// TwinCAT 3 PLC project NOTT_CRYO
// ProgramVersion: 3.1.4026.22
// CompilerDefines: VISU_USEPROPERTYINFO
// libraries:
//   ESO Cryo HMI Library, * (ESO)
//   ESO LDC Comm Common Library, * (ESO)
//   ESO LDC Comm Tcp Library, * (ESO)
//   ESO LDC Cryo Library, * (ESO)
//   METIS Cryo PLC, * (KU Leuven)
//   METIS Fuse Library, * (KU Leuven)
//   Tc2_ControllerToolbox, * (Beckhoff Automation GmbH)
//   Tc2_Standard, * (Beckhoff Automation GmbH)
//   Tc2_System, * (Beckhoff Automation GmbH)
//   Tc2_Utilities, * (Beckhoff Automation GmbH)
//   Tc3_EventLogger, * (Beckhoff Automation GmbH)
//   VisuDialogs
// project tree:
//   DUTs/Enumerations/CoolDOwn/ E_NOTT_CRYO_COOLDOWN_STATE.TcDUT
//   DUTs/Enumerations/WarmUP/ E_NOTT_CRYO_WARMUP_STATE.TcDUT
//   DUTs/Enumerations/ E_NOTT_CRYO_CTRL_CMD.TcDUT, E_NOTT_CRYO_CTRL_STATE.TcDUT, E_NOTT_CRYO_HEATER_CTRL.TcDUT
//   DUTs/Enumerations/TCtrl/ T_NOTT_CTRL_LOOP_CTRL.TcDUT
//   DUTs/Enumerations/TempVote/ E_ALL_NOTT_TEMPERATURES.TcDUT
//   DUTs/Structures/CoolDown/ T_NOTT_CRYO_COOLDOWN_CFG.TcDUT, T_NOTT_CRYO_COOLDOWN_CTRL.TcDUT, T_NOTT_CRYO_COOLDOWN_STAT.TcDUT
//   DUTs/Structures/Fan/ T_NOTT_FAN_CFG.TcDUT, T_NOTT_FAN_CTRL.TcDUT, T_NOTT_FAN_STAT.TcDUT
//   DUTs/Structures/Nott_Pump/rp/ T_NOTT_PUMPS_STAT.TcDUT, T_NOTT_PUMP_CFG.TcDUT
//   DUTs/Structures/Nott_Pump/tp/ T_NOTT_PUMP_HIPACE80_CFG.TcDUT, T_NOTT_PUMP_HIPACE80_STAT.TcDUT
//   DUTs/Structures/TempVote/ T_NOTT_TEMP_VOTE_CFG.TcDUT, T_NOTT_CRYO_TEMP_VOTE_STATUS.TcDUT
//   DUTs/Structures/ T_CRYO_EVAC_CFG_50.TcDUT, T_CRYO_EVAC_CTRL_50.TcDUT, T_CRYO_EVAC_STAT_50.TcDUT, T_NOTT_CRYO_CFG.TcDUT, T_NOTT_CRYO_CTRL.TcDUT, T_NOTT_CRYO_DEBUG.TcDUT, T_NOTT_CRYO_EVENTS.TcDUT, T_NOTT_CRYO_STAT.TcDUT, T_NOTT_CRYO_TRIGGERS.TcDUT
//   DUTs/Structures/WarmUp/ T_NOTT_CRYO_WARMUP_CFG.TcDUT, T_NOTT_CRYO_WARMUP_CTRL.TcDUT, T_NOTT_CRYO_WARMUP_STAT.TcDUT
//   / GlobalTextList.TcGTLO, PlcTask.TcTTO, Visualization Manager.TcVMO (not stored)
//   POUs/Devices/Control/ FB_NOTT_CTRL_TEMPERATURE.TcPOU, FB_NOTT_TCTRLs.TcPOU
//   POUs/Devices/Heaters/ FB_NOTT_HEATERS.TcPOU
//   POUs/Devices/Fans/ FB_NOTT_FAN.TcPOU
//   POUs/Devices/ThermalBox/ FB_NOTT_THERMAL_BOX_CONTROL.TcPOU
//   POUs/Devices/NOTT_Pump/Functions/ F_PfeifferExpoNewToLReal.TcPOU (not stored)
//   POUs/Devices/NOTT_Pump/rp/ FB_NOTT_PUMP_HICUBE_80_NEO.TcPOU (not stored)
//   POUs/Devices/NOTT_Pump/tp/ FB_NOTT_PUMP_HIPACE80.TcPOU (not stored)
//   POUs/Devices/Temperatures/ FB_NOTT_TEMPERATURES.TcPOU
//   POUs/Devices/Temp_voters/ FB_NOTT_VOTER.TcPOU, FB_NOTT_VOTERS.TcPOU, FB_NOTT_READ_WRITE_TEMP_VOTE_CONFIG.TcPOU
//   POUs/ FB_NOTT_CRYO_CTRL.TcPOU, MAIN.TcPOU
//   POUs/Routines/CoolDown/ FB_NOTT_CRYO_COOLDOWN.TcPOU
//   POUs/Routines/Evacuation/ FB_NOTT_CRYO_EVAC.TcPOU
//   POUs/Routines/WarmUp/ FB_NOTT_CRYO_WARMUP.TcPOU
//   VISUs/ GUI_TEMPLATE_HIPACE_80.TcVIS, TEMPLATE_NOTT_PUMPS.TcVIS, VISU_BASE_PLATE_HTR.TcVIS, VISU_Detector_Heater.TcVIS, VISU_NOTT_PRESSURES.TcVIS, VISU_NOTT_RP.TcVIS, VISU_NOTT_TP.TcVIS, VISU_PTC_COOLER.TcVIS
// real-time tasks:
//   TASK PlcTask: cycle T#10ms, priority 20, ADS port 350
// I/O:
//   DEVICE Device 1 (EtherCAT), AmsNetId 10.33.179.184.2.1
//     -A1 [EK1200-5000 EtherCAT Power supply (2A E-Bus)]
//       Term 2 (EL6070-0033) [EL6070-0033 1Ch. Licence key terminal, individual licences]
//       A1-N12 (EL4104) [EL4104 4Ch. Ana. Output 0-10V, 16bit]
//       Term 38 (EL2535) [EL2535 2Ch. Pulse Width Current Output (24V, 1A)]
//       Term 39 (EL1084) [EL1084 4Ch. Dig. Input 24V, 3ms, negative]
//       N15_RP_RS485 (EL6021) [EL6021 Interface (RS422/485)]
//       N16_TMP_RS485 (EL6021) [EL6021 Interface (RS422/485)]
//       A1-N5 (EL2068) [EL2068 8Ch. Dig Output 24V, 0.5A]
//       A1-N6_DET_HTR (EL9501) [EL9501 Power supply terminal 0...20 V DC, 0...2 A]
//       A1-N7_DET_SPR_HTR (EL9501) [EL9501 Power supply terminal 0...20 V DC, 0...2 A]
//       A1-N8_SIDECAR_HTR (EL9501) [EL9501 Power supply terminal 0...20 V DC, 0...2 A]
//       A1-N9_P_CHIP_HTR (EL9501) [EL9501 Power supply terminal 0...20 V DC, 0...2 A]
//       A1-N10 (EL2634) [EL2634 4Ch. Relay Output, NO (250V AC / 30V DC)]
//       A1-N11 (EL2634) [EL2634 4Ch. Relay Output, NO (250V AC / 30V DC)]
//       N17_Junction (EK1122) [EK1122 2 port EtherCAT junction]
//     -A2 [EK1101 EtherCAT Coupler (2A E-Bus, ID switch)]
//       A2-N3_T_Sidecar (EL3202-0010) [EL3202-0010 2Ch. Ana. Input PT100 (RTD), High Precision]
//       A2-N4_T_PhotoChip (EL3202-0010) [EL3202-0010 2Ch. Ana. Input PT100 (RTD), High Precision]
//       A2-N5_T_BasePlate (EL3202-0010) [EL3202-0010 2Ch. Ana. Input PT100 (RTD), High Precision]
//       A2-N6_T_Shield (EL3202-0010) [EL3202-0010 2Ch. Ana. Input PT100 (RTD), High Precision]
//       A2-N7_T_FF_Source (EL3202-0010) [EL3202-0010 2Ch. Ana. Input PT100 (RTD), High Precision]
//       A2-N8_T_Environment (EL3218) [EL3218-0000 8Ch. Ana. Input PT100 (RTD)]
//       A2-N9_FF_Current (EL4014) [EL4014 4Ch. Ana. Output 0-20mA, 12bit]
//       A2-N10 (EL3104) [EL3104 4Ch. Ana. Input +/-10V Diff.]
//       A2-N11 (EL3692) [EL3692 2Ch. resistance measurement terminal]
//       A2-N12_Fuse (EL9227-5500) [EL9227-5500 Overcurrent protection 24V DC, 2Ch., max. 10A (sum), adjustable, extended functionalities]
//       A2-N14_LS240 (EL6731) [EL6731 PROFIBUS DP Master]
//       A2-N15_24VPwr (EL9410) [EL9410 E-Bus Power Supplier  (Diagnostics)]
//       A2-N16 (EL1008) [EL1008 8Ch. Dig. Input 24V, 3ms]
//       A2-N17 (EL2612) [EL2612 2Ch. Relay Output, CO (125V AC / 30V DC)]
//       A2-N18_Pump_Start (EL2612) [EL2612 2Ch. Relay Output, CO (125V AC / 30V DC)]
//       A2-N19_PTC_RS485 (EL6021) [EL6021 Interface (RS422/485)]
//       A1-N17_BasePlate_Current_Monitor (EL3681) [EL3681 Digital multimeter terminal]
//       A1-N18_Shield_Current_Monitor (EL3681) [EL3681 Digital multimeter terminal]
//       Term 35 (EL9011) [EL9011 End Terminal]
//   DEVICE Device 6 (NOV-DP-RAM)
//   DEVICE LS240_Det_Temp_Sensors (EL6731), AmsNetId 10.33.179.184.3.1
//     Box 3 (GSD Box) (Model 240 Series) // Vendor: Lake Shore Cryotronics Revision: 1.0
// variable links:
//   NOTT_CRYO/NOTT_CRYO Instance <-> Device 1 (EtherCAT)/-A1/A1-N10 (EL2634)
//     PlcTask Inputs/MAIN.nott_cryo_ctrl.nott_heaters.h_detector.i_nCouplerState <-> InfoData/State
//     PlcTask Outputs/MAIN.nott_cryo_ctrl.nott_heaters.h_detector.io_el95x1.q_bEnable <-> Channel 1/Output
//     PlcTask Outputs/MAIN.nott_cryo_ctrl.nott_heaters.h_detector.io_el95x1.q_bEnable <-> Channel 2/Output
//     PlcTask Outputs/MAIN.nott_cryo_ctrl.nott_heaters.h_detector_spare.io_el95x1.q_bEnable <-> Channel 3/Output
//     PlcTask Outputs/MAIN.nott_cryo_ctrl.nott_heaters.h_detector_spare.io_el95x1.q_bEnable <-> Channel 4/Output
//   NOTT_CRYO/NOTT_CRYO Instance <-> Device 1 (EtherCAT)/-A1/A1-N11 (EL2634)
//     PlcTask Outputs/MAIN.nott_cryo_ctrl.nott_heaters.h_photonic_chip.io_el95x1.q_bEnable <-> Channel 3/Output
//     PlcTask Outputs/MAIN.nott_cryo_ctrl.nott_heaters.h_photonic_chip.io_el95x1.q_bEnable <-> Channel 4/Output
//     PlcTask Outputs/MAIN.nott_cryo_ctrl.nott_heaters.h_sidecar.io_el95x1.q_bEnable <-> Channel 1/Output
//     PlcTask Outputs/MAIN.nott_cryo_ctrl.nott_heaters.h_sidecar.io_el95x1.q_bEnable <-> Channel 2/Output
//   NOTT_CRYO/NOTT_CRYO Instance <-> Device 1 (EtherCAT)/-A1/A1-N12 (EL4104)
//     PlcTask Outputs/MAIN.nott_cryo_ctrl.nott_heaters.h_base_plate.io_cpau60.q_nSetVoltage <-> AO Output Channel 1/SetVoltage_BasePlate_HTR
//     PlcTask Outputs/MAIN.nott_cryo_ctrl.nott_heaters.h_shield.io_cpau60.q_nSetVoltage <-> AO Output Channel 2/SetVoltage_Shield_HTR
//   NOTT_CRYO/NOTT_CRYO Instance <-> Device 1 (EtherCAT)/-A1/A1-N5 (EL2068)
//     PlcTask Inputs/MAIN.nott_cryo_ctrl.evac.PVV1.Actuator.i_nCouplerState <-> InfoData/State
//     PlcTask Inputs/MAIN.nott_cryo_ctrl.nott_heaters.h_base_plate.i_nCouplerState <-> InfoData/State
//     PlcTask Inputs/MAIN.nott_cryo_ctrl.nott_heaters.h_shield.i_nCouplerState <-> InfoData/State
//     PlcTask Outputs/MAIN.nott_cryo_ctrl.evac.PVV1.Actuator.q_bCtrl <-> DOS Outputs Channel 4/PVV1_bCtrl
//     PlcTask Outputs/MAIN.nott_cryo_ctrl.evac.q_bPower_VAGC <-> DOS Outputs Channel 7/Output
//     PlcTask Outputs/MAIN.nott_cryo_ctrl.nott_heaters.h_base_plate.io_cpau60.q_bEnable <-> DOS Outputs Channel 1/bEnable_BasePlate_HTR
//     PlcTask Outputs/MAIN.nott_cryo_ctrl.nott_heaters.h_shield.io_cpau60.q_bEnable <-> DOS Outputs Channel 2/bEnable_Shield_HTR
//   NOTT_CRYO/NOTT_CRYO Instance <-> Device 1 (EtherCAT)/-A1/A1-N6_DET_HTR (EL9501)
//     PlcTask Inputs/MAIN.nott_cryo_ctrl.nott_heaters.h_detector.io_el95x1.i_bError <-> AO Output Status/Status/Error
//     PlcTask Inputs/MAIN.nott_cryo_ctrl.nott_heaters.h_detector.io_el95x1.i_bOutputOverload <-> AO Output Status/Status/Output Overload
//     PlcTask Inputs/MAIN.nott_cryo_ctrl.nott_heaters.h_detector.io_el95x1.i_bOverrange <-> AO Output Status/Status/Overrange
//     PlcTask Inputs/MAIN.nott_cryo_ctrl.nott_heaters.h_detector.io_el95x1.i_bUnderrange <-> AO Output Status/Status/Underrange
//     PlcTask Inputs/MAIN.nott_cryo_ctrl.nott_heaters.h_detector.io_el95x1.i_bWarning <-> AO Output Status/Status/Warning
//     PlcTask Inputs/MAIN.nott_cryo_ctrl.nott_heaters.h_detector.io_el95x1.i_rCurrent <-> AI Output Current Standard (Real32)/io_el95x1.i_rCurrent
//     PlcTask Inputs/MAIN.nott_cryo_ctrl.nott_heaters.h_detector.io_el95x1.i_rVoltage <-> AI Output Voltage Standard (Real32)/Value (Real32)
//     PlcTask Outputs/MAIN.nott_cryo_ctrl.nott_heaters.h_detector.io_el95x1.q_nOutputInterface <-> AO Output Standard (Real32)/Control/Output Interface
//     PlcTask Outputs/MAIN.nott_cryo_ctrl.nott_heaters.h_detector.io_el95x1.q_nOutputOperation <-> AO Output Standard (Real32)/Control/Output Operation
//     PlcTask Outputs/MAIN.nott_cryo_ctrl.nott_heaters.h_detector.io_el95x1.q_rSetVoltage <-> AO Output Standard (Real32)/Value (Real32)
//   NOTT_CRYO/NOTT_CRYO Instance <-> Device 1 (EtherCAT)/-A1/A1-N7_DET_SPR_HTR (EL9501)
//     PlcTask Inputs/MAIN.nott_cryo_ctrl.nott_heaters.h_detector_spare.i_nCouplerState <-> InfoData/State
//     PlcTask Inputs/MAIN.nott_cryo_ctrl.nott_heaters.h_detector_spare.io_el95x1.i_bError <-> AO Output Status/Status/Error
//     PlcTask Inputs/MAIN.nott_cryo_ctrl.nott_heaters.h_detector_spare.io_el95x1.i_bOutputOverload <-> AO Output Status/Status/Output Overload
//     PlcTask Inputs/MAIN.nott_cryo_ctrl.nott_heaters.h_detector_spare.io_el95x1.i_bOverrange <-> AO Output Status/Status/Overrange
//     PlcTask Inputs/MAIN.nott_cryo_ctrl.nott_heaters.h_detector_spare.io_el95x1.i_bUnderrange <-> AO Output Status/Status/Underrange
//     PlcTask Inputs/MAIN.nott_cryo_ctrl.nott_heaters.h_detector_spare.io_el95x1.i_bWarning <-> AO Output Status/Status/Warning
//     PlcTask Inputs/MAIN.nott_cryo_ctrl.nott_heaters.h_detector_spare.io_el95x1.i_rCurrent <-> AI Output Current Standard (Real32)/Value (Real32)
//     PlcTask Inputs/MAIN.nott_cryo_ctrl.nott_heaters.h_detector_spare.io_el95x1.i_rVoltage <-> AI Output Voltage Standard (Real32)/Value (Real32)
//     PlcTask Outputs/MAIN.nott_cryo_ctrl.nott_heaters.h_detector_spare.io_el95x1.q_nOutputInterface <-> AO Output Standard (Real32)/Control/Output Interface
//     PlcTask Outputs/MAIN.nott_cryo_ctrl.nott_heaters.h_detector_spare.io_el95x1.q_nOutputOperation <-> AO Output Standard (Real32)/Control/Output Operation
//     PlcTask Outputs/MAIN.nott_cryo_ctrl.nott_heaters.h_detector_spare.io_el95x1.q_rSetVoltage <-> AO Output Standard (Real32)/Value (Real32)
//   NOTT_CRYO/NOTT_CRYO Instance <-> Device 1 (EtherCAT)/-A1/A1-N8_SIDECAR_HTR (EL9501)
//     PlcTask Inputs/MAIN.nott_cryo_ctrl.nott_heaters.h_sidecar.i_nCouplerState <-> InfoData/State
//     PlcTask Inputs/MAIN.nott_cryo_ctrl.nott_heaters.h_sidecar.io_el95x1.i_bError <-> AO Output Status/Status/Error
//     PlcTask Inputs/MAIN.nott_cryo_ctrl.nott_heaters.h_sidecar.io_el95x1.i_bOutputOverload <-> AO Output Status/Status/Output Overload
//     PlcTask Inputs/MAIN.nott_cryo_ctrl.nott_heaters.h_sidecar.io_el95x1.i_bOverrange <-> AO Output Status/Status/Overrange
//     PlcTask Inputs/MAIN.nott_cryo_ctrl.nott_heaters.h_sidecar.io_el95x1.i_bUnderrange <-> AO Output Status/Status/Underrange
//     PlcTask Inputs/MAIN.nott_cryo_ctrl.nott_heaters.h_sidecar.io_el95x1.i_bWarning <-> AO Output Status/Status/Warning
//     PlcTask Inputs/MAIN.nott_cryo_ctrl.nott_heaters.h_sidecar.io_el95x1.i_rCurrent <-> AI Output Current Standard (Real32)/Value (Real32)
//     PlcTask Inputs/MAIN.nott_cryo_ctrl.nott_heaters.h_sidecar.io_el95x1.i_rVoltage <-> AI Output Voltage Standard (Real32)/Value (Real32)
//     PlcTask Outputs/MAIN.nott_cryo_ctrl.nott_heaters.h_sidecar.io_el95x1.q_nOutputInterface <-> AO Output Standard (Real32)/Control/Output Interface
//     PlcTask Outputs/MAIN.nott_cryo_ctrl.nott_heaters.h_sidecar.io_el95x1.q_nOutputOperation <-> AO Output Standard (Real32)/Control/Output Operation
//     PlcTask Outputs/MAIN.nott_cryo_ctrl.nott_heaters.h_sidecar.io_el95x1.q_rSetVoltage <-> AO Output Standard (Real32)/Value (Real32)
//   NOTT_CRYO/NOTT_CRYO Instance <-> Device 1 (EtherCAT)/-A1/A1-N9_P_CHIP_HTR (EL9501)
//     PlcTask Inputs/MAIN.nott_cryo_ctrl.nott_heaters.h_photonic_chip.i_nCouplerState <-> InfoData/State
//     PlcTask Inputs/MAIN.nott_cryo_ctrl.nott_heaters.h_photonic_chip.io_el95x1.i_bError <-> AO Output Status/Status/Error
//     PlcTask Inputs/MAIN.nott_cryo_ctrl.nott_heaters.h_photonic_chip.io_el95x1.i_bOutputOverload <-> AO Output Status/Status/Output Overload
//     PlcTask Inputs/MAIN.nott_cryo_ctrl.nott_heaters.h_photonic_chip.io_el95x1.i_bOverrange <-> AO Output Status/Status/Overrange
//     PlcTask Inputs/MAIN.nott_cryo_ctrl.nott_heaters.h_photonic_chip.io_el95x1.i_bUnderrange <-> AO Output Status/Status/Underrange
//     PlcTask Inputs/MAIN.nott_cryo_ctrl.nott_heaters.h_photonic_chip.io_el95x1.i_bWarning <-> AO Output Status/Status/Warning
//     PlcTask Inputs/MAIN.nott_cryo_ctrl.nott_heaters.h_photonic_chip.io_el95x1.i_rCurrent <-> AI Output Current Standard (Real32)/Value (Real32)
//     PlcTask Inputs/MAIN.nott_cryo_ctrl.nott_heaters.h_photonic_chip.io_el95x1.i_rVoltage <-> AI Output Voltage Standard (Real32)/Value (Real32)
//     PlcTask Outputs/MAIN.nott_cryo_ctrl.nott_heaters.h_photonic_chip.io_el95x1.q_nOutputInterface <-> AO Output Standard (Real32)/Control/Output Interface
//     PlcTask Outputs/MAIN.nott_cryo_ctrl.nott_heaters.h_photonic_chip.io_el95x1.q_nOutputOperation <-> AO Output Standard (Real32)/Control/Output Operation
//     PlcTask Outputs/MAIN.nott_cryo_ctrl.nott_heaters.h_photonic_chip.io_el95x1.q_rSetVoltage <-> AO Output Standard (Real32)/Value (Real32)
//   NOTT_CRYO/NOTT_CRYO Instance <-> Device 1 (EtherCAT)/-A1/N15_RP_RS485 (EL6021)
//     PlcTask Inputs/MAIN.nott_cryo_ctrl.evac.pump_pvp.comm.COMin_EL60xx/D[{0..21}] <-> COM TxPDO-Map Inputs/Data In {0..21}  (22 links)
//     PlcTask Inputs/MAIN.nott_cryo_ctrl.evac.pump_pvp.comm.COMin_EL60xx/Status <-> COM TxPDO-Map Inputs/Status
//     PlcTask Inputs/MAIN.nott_cryo_ctrl.evac.pump_pvp.comm.i_nCouplerState <-> InfoData/State
//     PlcTask Outputs/MAIN.nott_cryo_ctrl.evac.pump_pvp.comm.COMout_EL60xx/Ctrl <-> COM RxPDO-Map Outputs/Ctrl
//     PlcTask Outputs/MAIN.nott_cryo_ctrl.evac.pump_pvp.comm.COMout_EL60xx/D[{0..21}] <-> COM RxPDO-Map Outputs/Data Out {0..21}  (22 links)
//   NOTT_CRYO/NOTT_CRYO Instance <-> Device 1 (EtherCAT)/-A1/N16_TMP_RS485 (EL6021)
//     PlcTask Inputs/MAIN.nott_cryo_ctrl.evac.pump_tmp.comm.COMin_EL60xx/D[{0..21}] <-> COM TxPDO-Map Inputs/Data In {0..21}  (22 links)
//     PlcTask Inputs/MAIN.nott_cryo_ctrl.evac.pump_tmp.comm.COMin_EL60xx/Status <-> COM TxPDO-Map Inputs/Status
//     PlcTask Inputs/MAIN.nott_cryo_ctrl.evac.pump_tmp.comm.i_nCouplerState <-> InfoData/State
//     PlcTask Outputs/MAIN.nott_cryo_ctrl.evac.pump_tmp.comm.COMout_EL60xx/Ctrl <-> COM RxPDO-Map Outputs/Ctrl
//     PlcTask Outputs/MAIN.nott_cryo_ctrl.evac.pump_tmp.comm.COMout_EL60xx/D[{0..21}] <-> COM RxPDO-Map Outputs/Data Out {0..21}  (22 links)
//   NOTT_CRYO/NOTT_CRYO Instance <-> Device 1 (EtherCAT)/-A1/Term 39 (EL1084)
//     PlcTask Inputs/MAIN.nott_cryo_ctrl.bHMISwitch <-> Channel 2/Input
//   NOTT_CRYO/NOTT_CRYO Instance <-> Device 1 (EtherCAT)/-A2/A1-N17_BasePlate_Current_Monitor (EL3681)
//     PlcTask Inputs/MAIN.nott_cryo_ctrl.nott_heaters.h_base_plate.io_cpau60.i_nActCurrent <-> SAI Inputs/Value
//     PlcTask Inputs/MAIN.nott_cryo_ctrl.nott_heaters.h_base_plate.io_cpau60.i_nStatus <-> SAI Inputs/Status
//   NOTT_CRYO/NOTT_CRYO Instance <-> Device 1 (EtherCAT)/-A2/A1-N18_Shield_Current_Monitor (EL3681)
//     PlcTask Inputs/MAIN.nott_cryo_ctrl.nott_heaters.h_shield.io_cpau60.i_nActCurrent <-> SAI Inputs/Value
//     PlcTask Inputs/MAIN.nott_cryo_ctrl.nott_heaters.h_shield.io_cpau60.i_nStatus <-> SAI Inputs/Status
//   NOTT_CRYO/NOTT_CRYO Instance <-> Device 1 (EtherCAT)/-A2/A2-N10 (EL3104)
//     PlcTask Inputs/MAIN.nott_cryo_ctrl.nott_heaters.h_flat_field.io_flat_field.i_nActVoltage <-> AI Standard Channel 3/Value
//     PlcTask Inputs/MAIN.nott_cryo_ctrl.nott_heaters.h_flat_field.io_flat_field.i_nVoltageStatus <-> AI Standard Channel 3/Status
//     PlcTask Inputs/MAIN.nott_cryo_ctrl.sensor_HPG.i_nStatus <-> AI Standard Channel 2/Status
//     PlcTask Inputs/MAIN.nott_cryo_ctrl.sensor_HPG.i_nValue <-> AI Standard Channel 2/Value
//     PlcTask Inputs/MAIN.nott_cryo_ctrl.sensor_VAGC.i_nStatus <-> AI Standard Channel 1/Status
//     PlcTask Inputs/MAIN.nott_cryo_ctrl.sensor_VAGC.i_nValue <-> AI Standard Channel 1/Value
//   NOTT_CRYO/NOTT_CRYO Instance <-> Device 1 (EtherCAT)/-A2/A2-N16 (EL1008)
//     PlcTask Inputs/MAIN.nott_cryo_ctrl.evac.pump_pvp.i_bError <-> Channel 5/Input
//     PlcTask Inputs/MAIN.nott_cryo_ctrl.evac.pump_tmp.i_bError <-> Channel 8/Input
//     PlcTask Inputs/MAIN.nott_cryo_ctrl.evac.pump_tmp.i_bReady <-> Channel 7/Input
//   NOTT_CRYO/NOTT_CRYO Instance <-> Device 1 (EtherCAT)/-A2/A2-N17 (EL2612)
//     PlcTask Inputs/MAIN.nott_cryo_ctrl.cool_down.cooler.comm.i_nCouplerState <-> InfoData/State
//     PlcTask Outputs/MAIN.nott_cryo_ctrl.bHMIOutEnable <-> Channel 2/Output
//     PlcTask Outputs/MAIN.nott_cryo_ctrl.cool_down.cooler.q_bCtrlStart <-> Channel 1/Output
//   NOTT_CRYO/NOTT_CRYO Instance <-> Device 1 (EtherCAT)/-A2/A2-N18_Pump_Start (EL2612)
//     PlcTask Outputs/MAIN.nott_cryo_ctrl.evac.pump_pvp.q_bStart <-> Channel 1/RP_bEnable
//     PlcTask Outputs/MAIN.nott_cryo_ctrl.evac.pump_tmp.q_bStart <-> Channel 2/TP_bEnable
//   NOTT_CRYO/NOTT_CRYO Instance <-> Device 1 (EtherCAT)/-A2/A2-N19_PTC_RS485 (EL6021)
//     PlcTask Inputs/MAIN.nott_cryo_ctrl.cool_down.cooler.comm.COMin_EL60xx/D[{0..21}] <-> COM TxPDO-Map Inputs/Data In {0..21}  (22 links)
//     PlcTask Inputs/MAIN.nott_cryo_ctrl.cool_down.cooler.comm.COMin_EL60xx/Status <-> COM TxPDO-Map Inputs/Status
//     PlcTask Outputs/MAIN.nott_cryo_ctrl.cool_down.cooler.comm.COMout_EL60xx/Ctrl <-> COM RxPDO-Map Outputs/Ctrl
//     PlcTask Outputs/MAIN.nott_cryo_ctrl.cool_down.cooler.comm.COMout_EL60xx/D[{0..21}] <-> COM RxPDO-Map Outputs/Data Out {0..21}  (22 links)
//   NOTT_CRYO/NOTT_CRYO Instance <-> Device 1 (EtherCAT)/-A2/A2-N3_T_Sidecar (EL3202-0010)
//     PlcTask Inputs/MAIN.nott_cryo_ctrl.nott_temp.t_sidecar_1.i_nStatus <-> RTD Inputs Channel 1/Status
//     PlcTask Inputs/MAIN.nott_cryo_ctrl.nott_temp.t_sidecar_2.i_nStatus <-> RTD Inputs Channel 2/Status
//     PlcTask Inputs/MAIN.nott_cryo_ctrl.nott_temp.t_sidecar_1.i_nValue <-> RTD Inputs Channel 1/Value
//     PlcTask Inputs/MAIN.nott_cryo_ctrl.nott_temp.t_sidecar_2.i_nValue <-> RTD Inputs Channel 2/Value
//   NOTT_CRYO/NOTT_CRYO Instance <-> Device 1 (EtherCAT)/-A2/A2-N4_T_PhotoChip (EL3202-0010)
//     PlcTask Inputs/MAIN.nott_cryo_ctrl.nott_temp.t_photonic_chip_1.i_nStatus <-> RTD Inputs Channel 1/Status
//     PlcTask Inputs/MAIN.nott_cryo_ctrl.nott_temp.t_photonic_chip_2.i_nStatus <-> RTD Inputs Channel 2/Status
//     PlcTask Inputs/MAIN.nott_cryo_ctrl.nott_temp.t_photonic_chip_1.i_nValue <-> RTD Inputs Channel 1/Value
//     PlcTask Inputs/MAIN.nott_cryo_ctrl.nott_temp.t_photonic_chip_2.i_nValue <-> RTD Inputs Channel 2/Value
//   NOTT_CRYO/NOTT_CRYO Instance <-> Device 1 (EtherCAT)/-A2/A2-N5_T_BasePlate (EL3202-0010)
//     PlcTask Inputs/MAIN.nott_cryo_ctrl.nott_temp.t_base_plate_1.i_nStatus <-> RTD Inputs Channel 1/Status
//     PlcTask Inputs/MAIN.nott_cryo_ctrl.nott_temp.t_base_plate_2.i_nStatus <-> RTD Inputs Channel 2/Status
//     PlcTask Inputs/MAIN.nott_cryo_ctrl.nott_temp.t_base_plate_1.i_nValue <-> RTD Inputs Channel 1/Value
//     PlcTask Inputs/MAIN.nott_cryo_ctrl.nott_temp.t_base_plate_2.i_nValue <-> RTD Inputs Channel 2/Value
//   NOTT_CRYO/NOTT_CRYO Instance <-> Device 1 (EtherCAT)/-A2/A2-N6_T_Shield (EL3202-0010)
//     PlcTask Inputs/MAIN.nott_cryo_ctrl.nott_temp.t_shield_1.i_nStatus <-> RTD Inputs Channel 1/Status
//     PlcTask Inputs/MAIN.nott_cryo_ctrl.nott_temp.t_shield_2.i_nStatus <-> RTD Inputs Channel 2/Status
//     PlcTask Inputs/MAIN.nott_cryo_ctrl.nott_temp.t_shield_1.i_nValue <-> RTD Inputs Channel 1/Value
//     PlcTask Inputs/MAIN.nott_cryo_ctrl.nott_temp.t_shield_2.i_nValue <-> RTD Inputs Channel 2/Value
//   NOTT_CRYO/NOTT_CRYO Instance <-> Device 1 (EtherCAT)/-A2/A2-N7_T_FF_Source (EL3202-0010)
//     PlcTask Inputs/MAIN.nott_cryo_ctrl.nott_temp.t_flat_field_1.i_nStatus <-> RTD Inputs Channel 1/Status
//     PlcTask Inputs/MAIN.nott_cryo_ctrl.nott_temp.t_flat_field_2.i_nStatus <-> RTD Inputs Channel 2/Status
//     PlcTask Inputs/MAIN.nott_cryo_ctrl.nott_temp.t_flat_field_1.i_nValue <-> RTD Inputs Channel 1/Value
//     PlcTask Inputs/MAIN.nott_cryo_ctrl.nott_temp.t_flat_field_2.i_nValue <-> RTD Inputs Channel 2/Value
//   NOTT_CRYO/NOTT_CRYO Instance <-> Device 1 (EtherCAT)/-A2/A2-N8_T_Environment (EL3218)
//     PlcTask Inputs/MAIN.nott_cryo_ctrl.nott_temp.t_cabinet_1.i_nStatus <-> RTD Inputs Channel 5/Status
//     PlcTask Inputs/MAIN.nott_cryo_ctrl.nott_temp.t_cabinet_2.i_nStatus <-> RTD Inputs Channel 6/Status
//     PlcTask Inputs/MAIN.nott_cryo_ctrl.nott_temp.t_cabinet_1.i_nValue <-> RTD Inputs Channel 5/Value
//     PlcTask Inputs/MAIN.nott_cryo_ctrl.nott_temp.t_cabinet_2.i_nValue <-> RTD Inputs Channel 6/Value
//     PlcTask Inputs/MAIN.nott_cryo_ctrl.nott_temp.t_thermal_box_{1..4}.i_nStatus <-> RTD Inputs Channel {1..4}/Status  (4 links)
//     PlcTask Inputs/MAIN.nott_cryo_ctrl.nott_temp.t_thermal_box_{1..4}.i_nValue <-> RTD Inputs Channel {1..4}/Value  (4 links)
//   NOTT_CRYO/NOTT_CRYO Instance <-> Device 1 (EtherCAT)/-A2/A2-N9_FF_Current (EL4014)
//     PlcTask Inputs/MAIN.nott_cryo_ctrl.nott_heaters.h_flat_field.i_nCouplerState <-> InfoData/State
//     PlcTask Outputs/MAIN.nott_cryo_ctrl.nott_heaters.h_flat_field.io_flat_field.q_nSetCurrentCh{1..4} <-> AO Outputs Channel {1..4}/Analog output  (4 links)
//   NOTT_CRYO/NOTT_CRYO Instance <-> LS240_Det_Temp_Sensors (EL6731)/Box 3 (GSD Box) (Model 240 Series)
//     PlcTask Inputs/MAIN.nott_cryo_ctrl.nott_temp.t_detector.i_fValue <-> T_DET (Sensor Reading)/Inputs/Sensor Reading_0_0
//     PlcTask Inputs/MAIN.nott_cryo_ctrl.nott_temp.t_detector_spare.i_fValue <-> T_DET_SPARE (Sensor Reading)/Inputs/Sensor Reading_0_0
//   NOTT_CRYO/NOTT_CRYO Instance <-> NOTT_CRYO/NOTT_CRYO Instance
//     PlcTask Inputs/MAIN.nott_cryo_ctrl.evac.PVV1.Actuator.i_bOFF <-> PlcTask Outputs/MAIN.nott_cryo_ctrl.evac.q_bPVV1_OFF_Flag
//     PlcTask Inputs/MAIN.nott_cryo_ctrl.evac.PVV1.Actuator.i_bON <-> PlcTask Outputs/MAIN.nott_cryo_ctrl.evac.PVV1.Actuator.q_bCtrl
//     PlcTask Inputs/MAIN.nott_cryo_ctrl.evac.sensor_VAG1.i_nStatus <-> PlcTask Outputs/MAIN.nott_cryo_ctrl.evac.pump_pvp.q_nStatus
//     PlcTask Inputs/MAIN.nott_cryo_ctrl.evac.sensor_VAG1.i_nValue <-> PlcTask Outputs/MAIN.nott_cryo_ctrl.evac.pump_pvp.q_nValue
//     PlcTask Inputs/MAIN.nott_cryo_ctrl.nott_temp.t_base_plate_vote.i_bValid <-> PlcTask Outputs/MAIN.nott_cryo_ctrl.nott_voters.vote_base_plate.q_bValid
//     PlcTask Inputs/MAIN.nott_cryo_ctrl.nott_temp.t_base_plate_vote.i_lrValue <-> PlcTask Outputs/MAIN.nott_cryo_ctrl.nott_voters.vote_base_plate.q_lrTemp
//     PlcTask Inputs/MAIN.nott_cryo_ctrl.nott_temp.t_cabinet_vote.i_bValid <-> PlcTask Outputs/MAIN.nott_cryo_ctrl.nott_voters.vote_cabinet.q_bValid
//     PlcTask Inputs/MAIN.nott_cryo_ctrl.nott_temp.t_cabinet_vote.i_lrValue <-> PlcTask Outputs/MAIN.nott_cryo_ctrl.nott_voters.vote_cabinet.q_lrTemp
//     PlcTask Inputs/MAIN.nott_cryo_ctrl.nott_temp.t_detector_vote.i_bValid <-> PlcTask Outputs/MAIN.nott_cryo_ctrl.nott_voters.vote_detector.q_bValid
//     PlcTask Inputs/MAIN.nott_cryo_ctrl.nott_temp.t_detector_vote.i_lrValue <-> PlcTask Outputs/MAIN.nott_cryo_ctrl.nott_voters.vote_detector.q_lrTemp
//     PlcTask Inputs/MAIN.nott_cryo_ctrl.nott_temp.t_flat_field_vote.i_bValid <-> PlcTask Outputs/MAIN.nott_cryo_ctrl.nott_voters.vote_flat_field.q_bValid
//     PlcTask Inputs/MAIN.nott_cryo_ctrl.nott_temp.t_flat_field_vote.i_lrValue <-> PlcTask Outputs/MAIN.nott_cryo_ctrl.nott_voters.vote_flat_field.q_lrTemp
//     PlcTask Inputs/MAIN.nott_cryo_ctrl.nott_temp.t_master.i_bValid <-> PlcTask Outputs/MAIN.nott_cryo_ctrl.nott_voters.vote_master_temp.q_bValid
//     PlcTask Inputs/MAIN.nott_cryo_ctrl.nott_temp.t_master.i_lrValue <-> PlcTask Outputs/MAIN.nott_cryo_ctrl.nott_voters.vote_master_temp.q_lrTemp
//     PlcTask Inputs/MAIN.nott_cryo_ctrl.nott_temp.t_master_vot_1.i_bValid <-> PlcTask Outputs/MAIN.nott_cryo_ctrl.nott_voters.vote_master_1.q_bValid
//     PlcTask Inputs/MAIN.nott_cryo_ctrl.nott_temp.t_master_vot_2.i_bValid <-> PlcTask Outputs/MAIN.nott_cryo_ctrl.nott_voters.vote_master_2.q_bValid
//     PlcTask Inputs/MAIN.nott_cryo_ctrl.nott_temp.t_master_vot_1.i_lrValue <-> PlcTask Outputs/MAIN.nott_cryo_ctrl.nott_voters.vote_master_1.q_lrTemp
//     PlcTask Inputs/MAIN.nott_cryo_ctrl.nott_temp.t_master_vot_2.i_lrValue <-> PlcTask Outputs/MAIN.nott_cryo_ctrl.nott_voters.vote_master_2.q_lrTemp
//     PlcTask Inputs/MAIN.nott_cryo_ctrl.nott_temp.t_photonic_chip_vote.i_bValid <-> PlcTask Outputs/MAIN.nott_cryo_ctrl.nott_voters.vote_photonic_chip.q_bValid
//     PlcTask Inputs/MAIN.nott_cryo_ctrl.nott_temp.t_photonic_chip_vote.i_lrValue <-> PlcTask Outputs/MAIN.nott_cryo_ctrl.nott_voters.vote_photonic_chip.q_lrTemp
//     PlcTask Inputs/MAIN.nott_cryo_ctrl.nott_temp.t_shield_vote.i_bValid <-> PlcTask Outputs/MAIN.nott_cryo_ctrl.nott_voters.vote_shield.q_bValid
//     PlcTask Inputs/MAIN.nott_cryo_ctrl.nott_temp.t_shield_vote.i_lrValue <-> PlcTask Outputs/MAIN.nott_cryo_ctrl.nott_voters.vote_shield.q_lrTemp
//     PlcTask Inputs/MAIN.nott_cryo_ctrl.nott_temp.t_sidecar_vote.i_bValid <-> PlcTask Outputs/MAIN.nott_cryo_ctrl.nott_voters.vote_sidecar.q_bValid
//     PlcTask Inputs/MAIN.nott_cryo_ctrl.nott_temp.t_sidecar_vote.i_lrValue <-> PlcTask Outputs/MAIN.nott_cryo_ctrl.nott_voters.vote_sidecar.q_lrTemp
//     PlcTask Inputs/MAIN.nott_cryo_ctrl.nott_temp.t_thermal_box_vote.i_bValid <-> PlcTask Outputs/MAIN.nott_cryo_ctrl.nott_voters.vote_thermal_box.q_bValid
//     PlcTask Inputs/MAIN.nott_cryo_ctrl.nott_temp.t_thermal_box_vote.i_lrValue <-> PlcTask Outputs/MAIN.nott_cryo_ctrl.nott_voters.vote_thermal_box.q_lrTemp

CONFIGURATION NOTT_CRYO
    RESOURCE PLC ON TwinCAT3
        TASK PlcTask(INTERVAL := T#10ms, PRIORITY := 20);
        PROGRAM MAIN WITH PlcTask : MAIN;
    END_RESOURCE
END_CONFIGURATION

// ---- DUTs/Enumerations/CoolDOwn/E_NOTT_CRYO_COOLDOWN_STATE.TcDUT
{attribute 'qualified_only'}
{attribute 'strict'}
{attribute 'to_string'}
TYPE E_NOTT_CRYO_COOLDOWN_STATE :
(
	NONE := 0,							// Undefined state.
	OFF,								// Everything is OFF.
	START_PTC,							// Start Pulse Tube Cooler
	START_RAMPDOWN_DETECTOR,			// Start ramp down the detector temperature
	COOLING,
	OPERATIONAL_TEMPERATURE_ACHIEVED,
	STOP_COOLDOWN
	
);
END_TYPE

// ---- DUTs/Enumerations/WarmUP/E_NOTT_CRYO_WARMUP_STATE.TcDUT
{attribute 'qualified_only'}
{attribute 'strict'}
{attribute 'to_string'}
TYPE E_NOTT_CRYO_WARMUP_STATE :
(
    NONE := 0,                     // Undefined state.
    OFF,                           // Warm-up disabled.

    START_DETECTOR_PROTECTION,     // Enable detector heaters and temperature control.
    WAIT_DETECTOR_SAFE,            // Wait until detector is above the protection offset.

    START_WARMUP,                  // Enable remaining heaters.
    WARMING_UP,                    // Warm the cryostat.

    WARM_TEMPERATURE_ACHIEVED,     // All temperatures above warm threshold.

    STOP_WARMUP                    // Disable warm-up and return to OFF.
	
);
END_TYPE

// ---- DUTs/Enumerations/E_NOTT_CRYO_CTRL_CMD.TcDUT
{attribute 'qualified_only'}
{attribute 'strict'}
TYPE E_NOTT_CRYO_CTRL_CMD :
(
	NONE	:= 0,
	COOL,
	WARM_UP
);
END_TYPE

// ---- DUTs/Enumerations/E_NOTT_CRYO_CTRL_STATE.TcDUT
{attribute 'qualified_only'}
{attribute 'strict'}
TYPE E_NOTT_CRYO_CTRL_STATE :
(
	NONE 			:= 0,
	WARM_PRESS,				// Warm & Pressurized
	WARM_VACUUM,			// Warm & Vacuum
	COOLING_DOWN,			// Cooling down
	COLD,					// Cold, i.e. fully operational
	WARMING_UP,				// Warming up
	ERROR					// Controller failure
);
END_TYPE

// ---- DUTs/Enumerations/E_NOTT_CRYO_HEATER_CTRL.TcDUT
{attribute 'qualified_only'}
{attribute 'strict'}
TYPE E_NOTT_CRYO_HEATER_CTRL :
(
	NONE := 0,
	DET_IF, 
	COLD_PLATE,
	PREAMP
);
END_TYPE

// ---- DUTs/Enumerations/TCtrl/T_NOTT_CTRL_LOOP_CTRL.TcDUT
{attribute 'TcHmiSymbol.Show'}
TYPE T_NOTT_CTRL_LOOP_CTRL :
STRUCT
	    // general
   	{attribute 'TcHmiSymbol.Show'}
    eCtrlMode:      E_METIS_CTRL_MODE;  // AUTO or MANUAL
	{attribute 'TcHmiSymbol.Show'}	
    bEngMode:       BOOL;   // TRUE means engineering mode should be ON
	{attribute 'TcHmiSymbol.Show'}    
    bHold   : BOOL; // level-based
	{attribute 'TcHmiSymbol.Show'}    
    lrFixedSetpoint : LREAL;
	{attribute 'TcHmiSymbol.Show'}	
    lrSetpointOffset : LREAL;
    
    // 	
	//lrRampSetpointValue		: LREAL		:= 0.0;
	{attribute 'TcHmiSymbol.Show'}
	lrManualOut		: LREAL		:= 0.0;
   	{attribute 'TcHmiSymbol.Show'} 
    nInputTempIndex : INT;
	{attribute 'TcHmiSymbol.Show'}	
    nSetpointTempIndex : INT;
    
    // config reading/writing
	{attribute 'TcHmiSymbol.Show'}	
	bReadConfig         : BOOL;     // start reading the config file
	{attribute 'TcHmiSymbol.Show'}
	bWriteConfig        : BOOL;     // start writing the config file
    
    // output
	{attribute 'TcHmiSymbol.Show'}
    lrOutMaxLimit       : LREAL := 100.0;
	{attribute 'TcHmiSymbol.Show'}
    lrOutMinLimit       : LREAL := 0.0;
    
    // clear some diagnostics
    bClearForcedManualDiag : BOOL;
	{attribute 'TcHmiSymbol.Show'}
	eInputTempIndex:		 	E_ALL_NOTT_TEMPERATURES;
	{attribute 'TcHmiSymbol.Show'}
	eVariableSetpointIndex:		E_ALL_NOTT_TEMPERATURES;
END_STRUCT
END_TYPE

// ---- DUTs/Enumerations/TempVote/E_ALL_NOTT_TEMPERATURES.TcDUT
{attribute 'qualified_only'}
{attribute 'strict'}
{attribute 'to_string'}
TYPE E_ALL_NOTT_TEMPERATURES :
(

	empty_temp 				:= 0,	
	
	// SideCar (* 3 *)
	t_sidecar_1				:= 1,
	t_sidecar_2             := 2,
	t_sidecar_vote          := 3,
	// Photonic Chip (* 3 *)
	t_photonic_chip_1		:= 4,
	t_photonic_chip_2       := 5,
	t_photonic_chip_vote    := 6,
	// Base Plate (* 3 *)
	t_base_plate_1			:= 7,
	t_base_plate_2          := 8,
	t_base_plate_vote       := 9,
	// Shield (* 3 *)
	t_shield_1				:= 10,
	t_shield_2              := 11,
	t_shield_vote           := 12,	
	// Detector (* 3 *)
	t_detector				:= 13,
	t_detector_spare        := 14,
	t_detector_vote         := 15,
	// System temperatures   (* 3 *)
	// Legacy system-temperature channels; not used for cryostat state estimation.
	t_master				:= 16,
	t_master_vot_1          := 17,
	t_master_vot_2          := 18,
	// Flat Field   (* 3 *)
	t_flat_field_1			:= 19,
	t_flat_field_2          := 20,
	t_flat_field_vote       := 21,
	// Thermal Box   (* 5 *)
	t_thermal_box_1			:= 22,
	t_thermal_box_2         := 23,
	t_thermal_box_3			:= 24,
	t_thermal_box_4         := 25,
	t_thermal_box_vote      := 26,
	
		// Cabinet   (* 3 *)
	t_cabinet_1				:= 27,
	t_cabinet_2             := 28,
	t_cabinet_vote          := 29
	
);
END_TYPE

// ---- DUTs/Structures/CoolDown/T_NOTT_CRYO_COOLDOWN_CFG.TcDUT
TYPE T_NOTT_CRYO_COOLDOWN_CFG :
STRUCT	
	lrTemp_Det:				LREAL := 40.0;		// Detector target temperature [K]
	lrTemp_BasePlate:		LREAL := 100.0;		// Base plate target temperature [K]
	lrTemp_LowLimit:		LREAL := 73.0;		// Lowest temperature limit [K]
END_STRUCT
END_TYPE

// ---- DUTs/Structures/CoolDown/T_NOTT_CRYO_COOLDOWN_CTRL.TcDUT
TYPE T_NOTT_CRYO_COOLDOWN_CTRL :
STRUCT
	
	bEnable_Cooler:		BOOL := FALSE;
		// Command override (cor)
	cor_Cooler:				FB_CRYO_CMD_OVERRIDE;
END_STRUCT
END_TYPE

// ---- DUTs/Structures/CoolDown/T_NOTT_CRYO_COOLDOWN_STAT.TcDUT
TYPE T_NOTT_CRYO_COOLDOWN_STAT :
STRUCT
	{attribute 'TcHmiSymbol.Show'}
	{attribute 'TcHmiSymbol.ReadOnly'}
	bEnabled:		BOOL := FALSE;	// Controller active while bEnable is TRUE
	bConfigured:	BOOL := FALSE;	// Flag if controller has been configured.
	bError:			BOOL;			// Flag if controller is OK
	{attribute 'TcHmiSymbol.Show'}
	{attribute 'TcHmiSymbol.ReadOnly'}
	bActive:		BOOL;			// Flag if controller is ACTIVE
	bWarning:		BOOL := FALSE;	// Flag if there is a warning
	bEmergency:		BOOL := FALSE;	// Flag if there was Emergency valve closure
	bPTC_On:		BOOL;			// Flag if Prevacuum Pump is running
	bPTC_Ready:		BOOL;			// Flag if Prevacuum Pump is Ready
	{attribute 'TcHmiSymbol.Show'}
	{attribute 'TcHmiSymbol.ReadOnly'}
	bAlarm:			BOOL;
	{attribute 'TcHmiSymbol.Show'}
	{attribute 'TcHmiSymbol.ReadOnly'}
	bPressureAlarm:	BOOL := FALSE;
	{attribute 'TcHmiSymbol.Show'}
	{attribute 'TcHmiSymbol.ReadOnly'}
	bPumpAlarm:		BOOL := FALSE;


	// Generic controller OK flag.
	// Used for problems other than from the actuator.
	// This flag is used for problems coming from controllers
	// that extend the functionality of FB_CRYO_BIN_CTRL.
	bCtrlOK:	BOOL := TRUE;		

	nState:			E_NOTT_CRYO_COOLDOWN_STATE := E_NOTT_CRYO_COOLDOWN_STATE.NONE;
	
	sErrorText:		STRING(64);		// Error as text
	sState:			STRING(64);		// State as text
	{attribute 'TcHmiSymbol.Show'}
	{attribute 'TcHmiSymbol.ReadOnly'}
	sStatus:		STRING(64);		// Status as text
END_STRUCT
END_TYPE

// ---- DUTs/Structures/Fan/T_NOTT_FAN_CFG.TcDUT
TYPE T_NOTT_FAN_CFG :
STRUCT
	lrMinRunningDutyPct:	LREAL := 20.0;	// Minimum commanded running duty [%]
	lrMaxDutyPct:			LREAL := 100.0;	// Maximum commanded duty [%]
	lrStartDutyPct:		LREAL := 100.0;	// Startup boost duty [%]
	tStartBoost:			TIME := T#2S;
	tRpmWindow:			TIME := T#1S;
	tStallDelay:			TIME := T#5S;
	nPulsesPerRevolution:	UINT := 2;
	nPwmFullScale:			INT := 32767;	// EL2535 linked process-data full scale
	bInvertPwmOutput:		BOOL := FALSE;	// Set TRUE if the external interface inverts PWM
	bInvertTachInput:		BOOL := FALSE;	// Set TRUE if the ES1084 process bit is inverted
END_STRUCT
END_TYPE

// ---- DUTs/Structures/Fan/T_NOTT_FAN_CTRL.TcDUT
TYPE T_NOTT_FAN_CTRL :
STRUCT
	{attribute 'TcHmiSymbol.Show'}
	bEnable:			BOOL := FALSE;
	{attribute 'TcHmiSymbol.Show'}
	bAuto:				BOOL := TRUE;
	{attribute 'TcHmiSymbol.Show'}
	lrManualDutyPct:	LREAL := 0.0;
END_STRUCT
END_TYPE

// ---- DUTs/Structures/Fan/T_NOTT_FAN_STAT.TcDUT
TYPE T_NOTT_FAN_STAT :
STRUCT
	{attribute 'TcHmiSymbol.Show'}
	{attribute 'TcHmiSymbol.ReadOnly'}
	bActive:				BOOL := FALSE;
	{attribute 'TcHmiSymbol.Show'}
	{attribute 'TcHmiSymbol.ReadOnly'}
	bRunning:				BOOL := FALSE;
	{attribute 'TcHmiSymbol.Show'}
	{attribute 'TcHmiSymbol.ReadOnly'}
	bStallAlarm:			BOOL := FALSE;
	{attribute 'TcHmiSymbol.Show'}
	{attribute 'TcHmiSymbol.ReadOnly'}
	bTachMeasurementLimited:	BOOL := FALSE;
	{attribute 'TcHmiSymbol.Show'}
	{attribute 'TcHmiSymbol.ReadOnly'}
	lrDemandPct:			LREAL := 0.0;
	{attribute 'TcHmiSymbol.Show'}
	{attribute 'TcHmiSymbol.ReadOnly'}
	lrDutyPct:			LREAL := 0.0;
	{attribute 'TcHmiSymbol.Show'}
	{attribute 'TcHmiSymbol.ReadOnly'}
	lrSpeedRpm:			LREAL := 0.0;
	{attribute 'TcHmiSymbol.Show'}
	{attribute 'TcHmiSymbol.ReadOnly'}
	nPulseCount:			UDINT := 0;
	{attribute 'TcHmiSymbol.Show'}
	{attribute 'TcHmiSymbol.ReadOnly'}
	sName:				STRING(64);
	{attribute 'TcHmiSymbol.Show'}
	{attribute 'TcHmiSymbol.ReadOnly'}
	sAutoSetpointSource:	STRING(64);
END_STRUCT
END_TYPE

// ---- DUTs/Structures/Nott_Pump/rp/T_NOTT_PUMPS_STAT.TcDUT
TYPE T_NOTT_PUMPS_STAT EXTENDS T_CRYO_PUMP_BASE_STAT :
STRUCT


(*
Type:
0 - old bool: 0=FALSE, NOT 0 = TRUE.
1 - UDINT
2 - REAL * 100 (with leading zeros), e.g. 001571 corresponds with 15.71
4 - STRING (6)
7 - UINT (000 to 999)

INIT commands
312 Fw version Firmware version electronic drive unit 4 R
354 HW Version Hardware version electronic drive unit 4 R
399 NominalSpd Nominal rotation speed (rpm) 1 R rpm 0 999999

STATUS commands
010 Pumpg-Statn Pump 0 = off 1 = on 0 RW 0 1 0 x
060 CtrlViaInt Operation of the interface 
	1 = remote
	2 = RS-485
	4 = PV.can
	32 = Keys on the front panel

303 Error code Error code 4 R
	Err098 Internal communication error between interface board and drive
	Err117 Vacuum pump excess temperature (> 90 °C)
	Err174 Vacuum pump blocked
	Wrn117 High temperature vacuum pump (> 75 °C)

310 DrvCurrent Drive current 2 R A 0 9999.99
311 OpHrsPump Operating hours pump 1 R h 0 65535
313 DrvVoltage Drive voltage 2 R V 0 9999.99
316 *** DrvPower Drive power 1 R W 0 999999
330 TempPump Pump temperature 1 R °C 0 999999
398 ActualSpd Actual rotation speed (rpm) 1 R rpm 0 999999

*)

// INIT commands
	sFwVersion:		STRING(8);
	sHwVersion:		STRING(8);

// STATUS commands
	sFailureCode:	STRING(8) := 'OK';
	bTargetSpeed:	BOOL;		// Target Speed Reached
	nNominalSpeed:	DINT;		// [rpm] Nominal Pump Speed
	lrMotorVolt:	LREAL;		// Pump Motor Voltage [V]
	lrMotorCurr:	LREAL;		// Pump Motor Voltage [V]

	
	bFailure:		BOOL := FALSE;	// Err of Wrn (see cmd 303)
	nCtrlViaInt: DINT;
	sCtrlViaInt: STRING;
	
// Pressure Sensor
	// Init Commands
	
	PresSens_bSensorOn       : BOOL;
	PresSens_sSensorState    : STRING(8);

	PresSens_sFailureCode    : STRING(16);
	PresSens_bFailure        : BOOL;

	PresSens_sFwVersion      : STRING(16);
	PresSens_sHwVersion      : STRING(16);
	PresSens_sSerialNumber   : STRING(32);

	PresSens_sPressureRaw    : STRING(16);
	PresSens_lrPressure_hPa  : LREAL;
	PresSens_nPressure_hPa   : DINT;
	PresSens_sPressureText   : STRING(32);
	bGasBallastEnabled : BOOL;       // P050
	nGasBallastMode    : DINT;       // P068
	sGasBallastMode    : STRING(20); // Automatic / Closed / Open
	// Status Commands
END_STRUCT
END_TYPE

// ---- DUTs/Structures/Nott_Pump/rp/T_NOTT_PUMP_CFG.TcDUT
TYPE T_NOTT_PUMP_CFG  EXTENDS T_CRYO_PUMP_SERIAL_CFG:
STRUCT
	// HiCube 80 Neo specific command configuration.
// Pfeiffer Vacuum protocol for RS-485 interface.
// HiPace 80 Neo RS-485 device ID=1 (001) !!!
// MVP 015-2 RS-485 device ID=2 (002) !!!
// MPT 200 RS-485 device ID=8 (008) !!!

	// Definition of commands
	
// MVP 015-2 RS-485 device ID=2 (002) !!!
	C_CMD_NONE:				STRING(16) := '';
	C_CMD_sSetCtrlViaInt:	STRING(16) := '0021006003001';	// Control via DIO
	C_CMD_sCtrlViaInt:		STRING(16) := '0020006002=?';	//Read status Control via DIO
	
	C_CMD_nSpdSetMode:		STRING(16) := '0020002602=?';
	C_CMD_sFwVersion:		STRING(16) := '0020031202=?';
	C_CMD_sHwVersion:		STRING(16) := '0020035402=?';
	C_CMD_nNominalSpeed:	STRING(16) := '0020039902=?';
	C_CMD_bON:				STRING(16) := '0020001002=?';

	C_CMD_sErrorCode:		STRING(16) := '0020030302=?';
	C_CMD_nMotorCurr:		STRING(16) := '0020031002=?';
	C_CMD_nPumpHours:		STRING(16) := '0020031102=?';
	C_CMD_nMotorVolt:		STRING(16) := '0020031302=?';
	C_CMD_nElecPower:		STRING(16) := '0020031602=?';
	C_CMD_nPumpTemp:		STRING(16) := '0020033002=?';
	C_CMD_nPumpSpeed:		STRING(16) := '0020039802=?';
	C_CMD_bGasBallastOn: 	STRING(24) := '0021005006111111'; // P050 = ON
	C_CMD_bGasBallastOff: 	STRING(24) := '0021005006000000'; // P050 = OFF
	C_CMD_bGasBallast: 		STRING(16) := '0020005002=?';     // read P050
	C_CMD_bGasBallastAuto:  STRING(16) := '0021003003000';
	C_CMD_nGasBallastMode:  STRING(16) := '0020006802=?';
	
// MPT 200 RS-485 device ID=8 (008) !!!
	C_CMD_PresSens_bOn:				STRING(16) := '0080004102=?';
	C_CMD_PresSens_nErrorCode:		STRING(16) := '0080030302=?';
	C_CMD_PresSens_sSwVersion:		STRING(16) := '0080031202=?';
	C_CMD_PresSens_sHwVersion:		STRING(16) := '0080035402=?';
	C_CMD_PresSens_sSerialNum:		STRING(16) := '0080035502=?';
	C_CMD_PresSens_lrPressure:		STRING(16) := '0080074002=?';
	
	//C_CMD_sID000:			STRING(16) := '0001079706000001';	// Change all IDs to 1
	C_CMD_sID000:			STRING(16) := '';
	
END_STRUCT
END_TYPE

// ---- DUTs/Structures/Nott_Pump/tp/T_NOTT_PUMP_HIPACE80_CFG.TcDUT
TYPE T_NOTT_PUMP_HIPACE80_CFG EXTENDS T_CRYO_PUMP_SERIAL_CFG :
STRUCT
	// HIPACE80 specific command configuration.
// Pfeiffer Vacuum protocol for RS-485 interface.
// Assumed RS-485 device ID=1 (001) !!!

	// Definition of commands
	C_CMD_NONE:             	STRING(16) := '';
	
	C_CMD_sCtrlViaInt:      	STRING(16) := '0011006003001';   // write P060 = remote
	C_CMD_sFwVersion:       	STRING(16) := '0010031202=?';
	C_CMD_sHwVersion:       	STRING(16) := '0010035402=?';
	C_CMD_nNominalSpeed:    	STRING(16) := '0010039902=?';
	C_CMD_bDI1VentingEnable:	STRING(16) := '0011006203001';
	C_CMD_bDI1VentingDisable: 	STRING(16) := '0011001206000000';	
	C_CMD_bDI1Deactivated: 		STRING(16) := '0011006203000';   // disable vent DI
	C_CMD_nDI1Config : 			STRING(16) := '0010006202=?';    // Readback
	C_CMD_nRotSpdSwitch80 : 	STRING(16) := '0011030203080';  // Switch speed
	C_CMD_nRotSpdSwitchPt : 	STRING(16) := '0010070102=?';   // '0010030202=?';
	C_CMD_bVentEnable:			STRING(16) := '0010006202=?';
	C_CMD_bON:              	STRING(16) := '0010002302=?';       // MotorPump status
	// alternatively, if you want pumping station status:
	C_CMD_bPumpingStatn: STRING(16) := '0010001002=?';

	C_CMD_nCtrlMode:        STRING(16) := '0010006002=?';       // CtrlViaInt readback
	C_CMD_sErrorCode:       STRING(16) := '0010030302=?';
	C_CMD_bTargetSpeed:     STRING(16) := '0010030602=?';
	C_CMD_nMotorCurr:       STRING(16) := '0010031002=?';
	C_CMD_nPumpHours:       STRING(16) := '0010031102=?';
	C_CMD_nMotorVolt:       STRING(16) := '0010031302=?';
	C_CMD_nElecHours:       STRING(16) := '0010031402=?';
	C_CMD_nElecTemp:        STRING(16) := '0010032602=?';
	C_CMD_nPumpTemp:        STRING(16) := '0010033002=?';       // TempPmpBot
	C_CMD_nPumpSpeed:       STRING(16) := '0010039802=?';

	// optional extra, if useful:
	C_CMD_nRotorTemp:    STRING(16) := '0010038402=?';
	

END_STRUCT
END_TYPE

// ---- DUTs/Structures/Nott_Pump/tp/T_NOTT_PUMP_HIPACE80_STAT.TcDUT
TYPE T_NOTT_PUMP_HIPACE80_STAT EXTENDS T_CRYO_PUMP_HIPACE30_STAT :
STRUCT
	bPumpingStatn 	: BOOL;
	nRotorTemp    	: DINT;
	lrMotorCurr   	: LREAL;
	sCtrlViaInt   	: STRING(32);
	nCtrlViaInt   	: DINT;
	bVentEnable	  	: BOOL := TRUE;
	nRotSpdSwitchPt : DINT;
	
	nDI1Config      : DINT;        // raw DI1 config number
	bDI1Deactivated : BOOL;        // TRUE when P062 = 0
	bDI1Venting     : BOOL;        // TRUE when P062 = 1
	sDI1Config      : STRING(32);  // HMI text
END_STRUCT
END_TYPE

// ---- DUTs/Structures/TempVote/T_NOTT_TEMP_VOTE_CFG.TcDUT
TYPE T_NOTT_TEMP_VOTE_CFG :
STRUCT
	bEnabled        : BOOL;
    sDescription    : STRING; 

	sTemp1_Name	    : STRING;
	sTemp2_Name	    : STRING;
	sTemp3_Name	    : STRING;
	sTemp4_Name	    : STRING;
	sTemp5_Name	    : STRING;
	
	nVote_Method    : E_METIS_TEMP_VOTE_METHOD;
	
	eTemperature1   : E_ALL_NOTT_TEMPERATURES;
	eTemperature2   : E_ALL_NOTT_TEMPERATURES;
	eTemperature3   : E_ALL_NOTT_TEMPERATURES;
	eTemperature4   : E_ALL_NOTT_TEMPERATURES;
	eTemperature5   : E_ALL_NOTT_TEMPERATURES;
END_STRUCT
END_TYPE

// ---- DUTs/Structures/TempVote/T_NOTT_CRYO_TEMP_VOTE_STATUS.TcDUT
TYPE T_NOTT_CRYO_TEMP_VOTE_STATUS:
STRUCT
		//
	// Status coming from the analog input terminal.
	// This is nothing to do with the sensor, i.e. the reading can be
	// inside the input terminal measuring range but still it might
	// not be inside the sensor measuring range!
	//
	bInputUnder:		BOOL;
	bInputOver:			BOOL;
	bInputError:		BOOL;
	bInputToggle:		BOOL;
	bInputValid:		BOOL;
	bInputActive:		BOOL	:= FALSE;
	nRawValue:			INT;

	// Calculated status of the sensor
	bError:				BOOL;
	
	{attribute 'TcHmiSymbol.Show'}
	{attribute 'TcHmiSymbol.ReadOnly'}
	lrRamp:		LREAL;	// Temperature ramp [deg/min]
	
	{attribute 'TcHmiSymbol.Show'}

	bSimulated:		BOOL;				// Flag indicating if the value is simulated.
	{attribute 'TcHmiSymbol.Show'}

	lrSimTempK:	LREAL;				// Simulated Temp [K]

	{attribute 'TcHmiSymbol.Show'}

	bEnabled:		BOOL	:= FALSE;	// Flag indicating if the voter is enabled
    
	{attribute 'TcHmiSymbol.Show'}

	sDescription:	STRING;	// User description of the voter (e.g. 'Average detector T')
    
	{attribute 'TcHmiSymbol.Show'}

	bValid:			BOOL	:= FALSE;	// Flag indicating if the value is valid.
	{attribute 'TcHmiSymbol.Show'}
	{attribute 'TcHmiSymbol.ReadOnly'}
	lrTempK:		LREAL;				// Calculated Temperature in K
	sStatus:		STRING;				// Status string

	// Flags indicating connected sensor is Valid.
	{attribute 'TcHmiSymbol.Show'}
	{attribute 'TcHmiSymbol.ReadOnly'}
	lrSens1TempK:		LREAL;
	{attribute 'TcHmiSymbol.Show'}
	{attribute 'TcHmiSymbol.ReadOnly'}
	lrSens2TempK:		LREAL;
	{attribute 'TcHmiSymbol.Show'}
	{attribute 'TcHmiSymbol.ReadOnly'}
	lrSens3TempK:		LREAL;
	{attribute 'TcHmiSymbol.Show'}
	{attribute 'TcHmiSymbol.ReadOnly'}
	lrSens4TempK:		LREAL;
	{attribute 'TcHmiSymbol.Show'}
	{attribute 'TcHmiSymbol.ReadOnly'}
	lrSens5TempK:		LREAL;
	
	{attribute 'TcHmiSymbol.Show'}
	{attribute 'TcHmiSymbol.ReadOnly'}
	bValidSensor1:		BOOL	:= FALSE;
	{attribute 'TcHmiSymbol.Show'}
	{attribute 'TcHmiSymbol.ReadOnly'}
	bValidSensor2:		BOOL	:= FALSE;
	{attribute 'TcHmiSymbol.Show'}
	{attribute 'TcHmiSymbol.ReadOnly'}
	bValidSensor3:		BOOL	:= FALSE;
	{attribute 'TcHmiSymbol.Show'}
	{attribute 'TcHmiSymbol.ReadOnly'}
	bValidSensor4:		BOOL	:= FALSE;
	{attribute 'TcHmiSymbol.Show'}
	{attribute 'TcHmiSymbol.ReadOnly'}
	bValidSensor5:		BOOL	:= FALSE;
	{attribute 'TcHmiSymbol.ShowRecursively'}

	stAlarms:		T_CRYO_ALARMS;	

	bInRange:		BOOL	:= FALSE;

	lrTempC:		LREAL;				// Temp [deg C]
	
	{attribute 'TcHmiSymbol.Show'}
	aTempIndexes:		ARRAY[0..4] OF E_ALL_NOTT_TEMPERATURES;
	{attribute 'TcHmiSymbol.Show'}
	nVoteMethod:		E_METIS_TEMP_VOTE_METHOD;

    //bEnabled:       BOOL;	
	
END_STRUCT
END_TYPE

// ---- DUTs/Structures/T_CRYO_EVAC_CFG_50.TcDUT
TYPE T_CRYO_EVAC_CFG_50 :
STRUCT
	// Pressure sensor gauge types
	nType_VAG1:		E_CRYO_SENSOR_TYPE_PRESS := E_CRYO_SENSOR_TYPE_PRESS.PKR_360;
	nType_VAGC:		E_CRYO_SENSOR_TYPE_PRESS := E_CRYO_SENSOR_TYPE_PRESS.PKR_360;

	// Thresholds
	lrThld_TMP_before_PVV1:	LREAL := 0.01;	// Cryo pressure threshold to start TMP before opening PVV1 [mbar] 
	lrThld_TMP_after_PVV1:	LREAL := 0.1;	// Cryo pressure threshold to start TMP after opening PVV1 [mbar] 
	lrThld_Prevacuum:		LREAL := 5.0;	// Prevacuum pressure threshold [mbar]
	lrThld_Vacuum:			LREAL := 0.0001;// At this Cryo pressure evacuation has started [mbar]
	
	tDelayAfterClosingValves:		TIME := T#3S;	// Delay after closing all valves before stopping Pumps
END_STRUCT
END_TYPE

// ---- DUTs/Structures/T_CRYO_EVAC_CTRL_50.TcDUT
TYPE T_CRYO_EVAC_CTRL_50 :
STRUCT
	//
	// Enable flags
	//
	
	// Flags for control of pumps.
	// Seeting the flag to TRUE  will start the pump.
	// Seeting the flag to FALSE will stop  the pump.
	bEnable_PVP:	BOOL := FALSE;	// Prevacuum pump
	bEnable_TMP:	BOOL := FALSE;	// Turbo molecular pump
	
	// Flags for control of valves
	// Seeting the flag to TRUE  will open  the valve.
	// Seeting the flag to FALSE will close the valve.
	bEnable_PVV1:	BOOL := FALSE;
	
	
	//
	// Override flags
	//
	
	// Valve command override handling
	cor_PVV1:	FB_CRYO_CMD_OVERRIDE;

	// Pumps command override handling.
	cor_PVP:	FB_CRYO_CMD_OVERRIDE;
	cor_TMP:	FB_CRYO_CMD_OVERRIDE;

	// Pressure Simulation override
	por_VAG1:	FB_CRYO_CMD_OVERRIDE;
	

	//
	// Simulation flags.
	// NOTE: This is only needed for the total simulation
	//       of the system that is normally done in Control Model.
	//
	bSim_Press_VAG1:	BOOL;
	
END_STRUCT
END_TYPE

// ---- DUTs/Structures/T_CRYO_EVAC_STAT_50.TcDUT
TYPE T_CRYO_EVAC_STAT_50 :
STRUCT
	bEnabled:		BOOL := FALSE;	// Controller active while bEnable is TRUE
	bConfigured:	BOOL := FALSE;	// Flag if controller has been configured.
	bError:			BOOL;			// Flag if controller is OK
	bActive:		BOOL;			// Flag if controller is ACTIVE
	bWarning:		BOOL := FALSE;	// Flag if there is a warning
	bEmergency:		BOOL := FALSE;	// Flag if there was Emergency valve closure
	bPVP_On:		BOOL;			// Flag if Prevacuum Pump is running
	bPVP_Ready:		BOOL;			// Flag if Prevacuum Pump is Ready
	bTMP_On:		BOOL;			// Flag if Turbo Molecular Pump is running
	bTMP_Ready:		BOOL;			// Flag if Turbo Molecular Pump is Ready

	// Generic controller OK flag.
	// Used for problems other than from the actuator.
	// This flag is used for problems coming from controllers
	// that extend the functionality of FB_CRYO_BIN_CTRL.
	bCtrlOK:	BOOL := TRUE;		

	nState:			E_CRYO_EVAC_STATE_50	:= E_CRYO_EVAC_STATE_50.NONE;
	
	sErrorText:		STRING(64);		// Error as text
	sState:			STRING(64);		// State as text
	{attribute 'TcHmiSymbol.Show'}
	{attribute 'TcHmiSymbol.ReadOnly'}
	sStatus:		STRING(64);		// Status as text
END_STRUCT
END_TYPE

// ---- DUTs/Structures/T_NOTT_CRYO_CFG.TcDUT
TYPE T_NOTT_CRYO_CFG :
STRUCT
	lrTemp_Warm:			LREAL := 293.0;		// Warm temperature limit [K] = 20 C
	lrTemp_Warm_Reset:	LREAL := 295.0;		// Cold-status reset threshold [K]
	
	
	lrTemp_Sidecar:			LREAL := 120.0;		// Heater preamp target temperature [K]
	lrTemp_DET_Target:		LREAL :=  40.0;		// Target Detector Interface temperature [K]
	lrTemp_BasePlate_OP:	LREAL := 100.0;		// Operational base plate temperature limit [K]
	lrTemp_DET_OP_Reset:	LREAL :=  42.0;		// Detector operational reset threshold [K]
	lrTemp_BasePlate_OP_Reset: LREAL := 105.0;	// Base plate operational reset threshold [K]
	lrTemp_LowLimit:		LREAL :=  40.0;		// Lowest temperature limit [K]
	

	lrPress_Atm:			LREAL := 700.0;		// Atmospheric pressure limit   [mbar]
	lrPress_InVac:			LREAL := 10.0E-1;	// In vacuum limit   [mbar]
	lrPress_InVac_Reset:	LREAL := 12.0E-1;	// In-vacuum reset threshold [mbar]
	lrPress_GoodVac:		LREAL := 10.0E-4;	// Good Vacuum limit [mbar]
	lrPress_GoodVac_Reset:	LREAL := 20.0E-4;	// Good-vacuum reset threshold [mbar]
	lrPress_OP:			LREAL := 10.0E-5;	// Operational pressure limit [mbar]
	lrPress_OP_Reset:		LREAL := 20.0E-5;	// Operational pressure reset threshold [mbar]
	

END_STRUCT
END_TYPE

// ---- DUTs/Structures/T_NOTT_CRYO_CTRL.TcDUT
TYPE T_NOTT_CRYO_CTRL :
STRUCT
	bExecute:	BOOL := FALSE;
	nCommand:	E_NOTT_CRYO_CTRL_CMD := E_NOTT_CRYO_CTRL_CMD.NONE;
	
	bReset:		BOOL := FALSE;		// RESET Command

	// Command to repressurize the system. 
	// Exists only in full simulation in order to bring the 
	// system to atmospheric pressure.
	// In reality, repressurization is done by opening a manual valve.
	bSim_Repress:	BOOL := FALSE;	

	//
	// Enable flags used to activate system functions. 	
	//
	{attribute 'TcHmiSymbol.Show'}
	bEnable_Evac:		BOOL := FALSE;
	{attribute 'TcHmiSymbol.Show'}	
	bEnable_CoolDown:		BOOL := FALSE;	
	
	//bEnable_Coole:		BOOL := FALSE;
	bEnable_Heater:	BOOL := FALSE;
	{attribute 'TcHmiSymbol.Show'}	
	bEnable_WarmUp:		BOOL := FALSE;

	//	
	// Safe flags saying what is safe and what not.
	//
	bSafe_Cooling:		BOOL := FALSE;
	bSafe_Warmup:		BOOL := FALSE;

	//
	// Simulation flags.
	//
	
	// Pressure Simulation flags
	bSim_Press_VAGC:	BOOL := FALSE;
	bSim_Press_HPG:		BOOL := FALSE;


	//
	// System overrides for commands and sensor readings.
	//	
	// Command override (cor)
	cor_WarmUp:			FB_CRYO_CMD_OVERRIDE;
	cor_CoolDown:			FB_CRYO_CMD_OVERRIDE;
	cor_Evac:				FB_CRYO_CMD_OVERRIDE;
	cor_Heater_IF:			FB_CRYO_CMD_OVERRIDE;
	cor_Heater_Preamp:		FB_CRYO_CMD_OVERRIDE;
	cor_Heater_ColdPlate:	FB_CRYO_CMD_OVERRIDE;

	// Temperature Simulation override (tor)
	tor_Ambient:			FB_CRYO_CMD_OVERRIDE;
	tor_DetMon:				FB_CRYO_CMD_OVERRIDE;
	tor_ColdPlate:			FB_CRYO_CMD_OVERRIDE;
	tor_WarmFlange:			FB_CRYO_CMD_OVERRIDE;
	tor_WarmOptics:			FB_CRYO_CMD_OVERRIDE;
	tor_LS336:				FB_CRYO_CMD_OVERRIDE;

	// Pressure Simulation override (por)
	por_VAGC:				FB_CRYO_CMD_OVERRIDE;
	por_HPG:				FB_CRYO_CMD_OVERRIDE;


	
	// Lakeshore related control parameters
	bLS_UpdateSETP:		BOOL := FALSE;	// If TRUE, this flag will trigger Lakeshore SETP.
	lrLS_SETP:			LREAL := 40.0;	// New SETP
	lrLS_RAMP:			LREAL := 0.5;	// RAMP [K/min]
	
END_STRUCT
END_TYPE

// ---- DUTs/Structures/T_NOTT_CRYO_DEBUG.TcDUT
TYPE T_NOTT_CRYO_DEBUG :
STRUCT
	nCycleCounter:	UDINT := 0;
END_STRUCT
END_TYPE

// ---- DUTs/Structures/T_NOTT_CRYO_EVENTS.TcDUT
TYPE T_NOTT_CRYO_EVENTS :
STRUCT
	info:		FB_TcMessage;
	warning:	FB_TcMessage;
	error:		FB_TcAlarm;
	critical:	FB_TcAlarm;
	
END_STRUCT
END_TYPE

// ---- DUTs/Structures/T_NOTT_CRYO_STAT.TcDUT
TYPE T_NOTT_CRYO_STAT :
STRUCT
	//
	// Common attributes
	//
	bConfigured:	BOOL := FALSE;
	bSystemStarted:	BOOL := FALSE;	// Indicates if M_GetState has been called.

	bDone:			BOOL;			// Flag if controller is OK
	bBusy:			BOOL;			// Flag if controller is BUSY
	bError:			BOOL;			// Flag if controller is OK
	bActive:		BOOL;			// Flag if controller is ACTIVE
	
	nLastCommand:	E_NOTT_CRYO_CTRL_CMD 	:= E_NOTT_CRYO_CTRL_CMD.NONE;
	nState:			E_NOTT_CRYO_CTRL_STATE	:= E_NOTT_CRYO_CTRL_STATE.NONE;
	{attribute 'TcHmiSymbol.Show'}
	{attribute 'TcHmiSymbol.ReadOnly'}
	sState:			STRING(64);		// State as text


	//
	// PDS Cryo Controller specific attributes
	//
	
	// Simulation
	bSimulation:	BOOL := FALSE;	// If TRUE, System is simulated - Variant (V2_SIM)	
	bSim_RepressEnabled:	BOOL := FALSE;
	{attribute 'TcHmiSymbol.Show'}
	{attribute 'TcHmiSymbol.ReadOnly'}
	bVacuum:		BOOL := FALSE;
	{attribute 'TcHmiSymbol.Show'}
	{attribute 'TcHmiSymbol.ReadOnly'}		
	bVacuumOK:		BOOL := FALSE;		
	{attribute 'TcHmiSymbol.Show'}
	{attribute 'TcHmiSymbol.ReadOnly'}
	bPressureValid:	BOOL := FALSE;
	{attribute 'TcHmiSymbol.Show'}
	{attribute 'TcHmiSymbol.ReadOnly'}
	lrPressure_mbar:	LREAL;
	{attribute 'TcHmiSymbol.Show'}
	{attribute 'TcHmiSymbol.ReadOnly'}
	bCold:			BOOL := FALSE;	// Detector vote < cfg.lrTemp_Warm and cryostat is in vacuum
	{attribute 'TcHmiSymbol.Show'}
	{attribute 'TcHmiSymbol.ReadOnly'}
	bOP:			BOOL := FALSE;	// Detector/base-plate temperatures and VAGC pressure are operational

	bCoolantFlowOK:	BOOL := FALSE;		
	{attribute 'TcHmiSymbol.Show'}
	{attribute 'TcHmiSymbol.ReadOnly'}
	bHighestTempValid:	BOOL := FALSE;	// Highest temperature Valid flag
	{attribute 'TcHmiSymbol.Show'}
	{attribute 'TcHmiSymbol.ReadOnly'}
	bLowestTempValid:	BOOL := FALSE;	// Lowest temperature Valid flag
	{attribute 'TcHmiSymbol.Show'}
	{attribute 'TcHmiSymbol.ReadOnly'}
	lrHighestTempK:	LREAL;	// Highest temperature [K] in Cryostat
	{attribute 'TcHmiSymbol.Show'}
	{attribute 'TcHmiSymbol.ReadOnly'}
	lrLowestTempK:	LREAL;	// Lowest temperature [K] in Cryostat
	{attribute 'TcHmiSymbol.Show'}
	{attribute 'TcHmiSymbol.ReadOnly'}
	sLowestTempName:	STRING;
	{attribute 'TcHmiSymbol.Show'}
	{attribute 'TcHmiSymbol.ReadOnly'}
	sHighestTempName:	STRING;
	
	bIsPVPRunning:		BOOL := FALSE;
	bIsTMPRunning:		BOOL := FALSE;

END_STRUCT
END_TYPE

// ---- DUTs/Structures/T_NOTT_CRYO_TRIGGERS.TcDUT
TYPE T_NOTT_CRYO_TRIGGERS :
STRUCT
	//
	// Evacuation pumps
	//
	PVV1_Open:		R_TRIG;	// evac.PVV1.in_bEnable
	PVV1_Close:		F_TRIG;	// evac.PVV1.in_bEnable
	PVV1_Opened:	R_TRIG;	// evac.PVV1.stat.bActON
	PVV1_Closed:	R_TRIG;	// evac.PVV1.stat.bActOFF

	PVP_Start:		R_TRIG;	// evac.pump_pvp.in_bEnable
	PVP_Stop:		F_TRIG;	// evac.pump_pvp.in_bEnable
	PVP_Ready:		R_TRIG;	// evac.pump_pvp.stat.bReady
	PVP_Stopped:	F_TRIG;	// evac.pump_pvp.stat.bMoving

	//
	// Evacuation valve
	//
	TMP_Start:		R_TRIG;	// evac.pump_tmp.in_bEnable
	TMP_Stop:		F_TRIG;	// evac.pump_tmp.in_bEnable
	TMP_Ready:		R_TRIG;	// evac.pump_tmp.stat.bReady
	TMP_Stopped:	F_TRIG;	// evac.pump_tmp.stat.bMoving
	
	//
	// Heaters
	//
	Heater_DetIF_Enable:		R_TRIG;	// Heater_DetIF.in_bEnable
	Heater_DetIF_Disable:		F_TRIG;	// Heater_DetIF.in_bEnable
	Heater_DetIF_ON:			R_TRIG;	// Heater_DetIF.stat.bActON
	Heater_DetIF_OFF:			R_TRIG;	// Heater_DetIF.stat.bActOFF

	Heater_Preamp_Enable:		R_TRIG;	// Heater_Preamp.in_bEnable
	Heater_Preamp_Disable:		F_TRIG;	// Heater_Preamp.in_bEnable
	Heater_Preamp_ON:			R_TRIG;	// Heater_Preamp.stat.bActON
	Heater_Preamp_OFF:			R_TRIG;	// Heater_Preamp.stat.bActOFF

	Heater_ColdPlate_Enable:	R_TRIG;	// Heater_ColdPlate.in_bEnable
	Heater_ColdPlate_Disable:	F_TRIG;	// Heater_ColdPlate.in_bEnable
	Heater_ColdPlate_ON:		R_TRIG;	// Heater_ColdPlate.stat.bActON
	Heater_ColdPlate_OFF:		R_TRIG;	// Heater_ColdPlate.stat.bActOFF

	//
	// Cooler
	//
	Cooler_Enable:		R_TRIG;	// cooler.in_bEnable
	Cooler_Disable:		F_TRIG;	// cooler.in_bEnable
	Cooler_ON:			R_TRIG;	// cooler.stat.nDevState
	Cooler_OFF:			R_TRIG;	// cooler.stat.nDevState


	//
	// Pressure and Temperature status flags
	//
	
	// Vacuum
	Vacuum_ON:		R_TRIG;	// stat.bInVacuum
	Vacuum_OFF:		F_TRIG;	// stat.bInVacuum
	Vacuum_OK:		R_TRIG;	// stat.bGoodVacuum
	Vacuum_NOT_OK:	F_TRIG;	// stat.bGoodVacuum

	// Temperature
	Cold_ON:		R_TRIG;	// stat.bCold
	Cold_OFF:		F_TRIG;	// stat.bCold
	OP_ON:			R_TRIG;	// stat.bOP
	OP_OFF:			F_TRIG;	// stat.bOP
	
END_STRUCT
END_TYPE

// ---- DUTs/Structures/WarmUp/T_NOTT_CRYO_WARMUP_CFG.TcDUT
TYPE T_NOTT_CRYO_WARMUP_CFG :
STRUCT

	
	lrTemp_Det_OffSet:		LREAL := 25.0;	// Detector offset temperature before remaing heaters are turned ON [K]
	lrTemp_Det:				LREAL := 300.0;		// Detector target temperature [K]
	lrTemp_BasePlate:		LREAL := 300.0;		// Base plate target temperature [K]
	lrTemp_Shield:			LREAL := 300.0;		// Base plate target temperature [K]
	lrTemp_Sidecar:		    LREAL := 300.0;		// Base plate target temperature [K]
	lrTemp_FlatField:		LREAL := 300.0;		// Base plate target temperature [K]
	lrTemp_PhotonicChip: 	LREAL := 300.0;
		
	lrTemp_HighLimit:		LREAL := 305.0;		// Highest temperature limit [K]
END_STRUCT
END_TYPE

// ---- DUTs/Structures/WarmUp/T_NOTT_CRYO_WARMUP_CTRL.TcDUT
TYPE T_NOTT_CRYO_WARMUP_CTRL :
STRUCT
	

END_STRUCT
END_TYPE

// ---- DUTs/Structures/WarmUp/T_NOTT_CRYO_WARMUP_STAT.TcDUT
TYPE T_NOTT_CRYO_WARMUP_STAT :
STRUCT
	{attribute 'TcHmiSymbol.Show'}
	{attribute 'TcHmiSymbol.ReadOnly'}
	bEnabled:		BOOL := FALSE;	// Controller active while bEnable is TRUE
	bConfigured:	BOOL := FALSE;	// Flag if controller has been configured.
	bError:			BOOL;			// Flag if controller is OK
	{attribute 'TcHmiSymbol.Show'}
	{attribute 'TcHmiSymbol.ReadOnly'}
	bActive:		BOOL;			// Flag if controller is ACTIVE
	bWarning:		BOOL := FALSE;	// Flag if there is a warning
	bEmergency:		BOOL := FALSE;	// Flag if there was Emergency valve closure
	{attribute 'TcHmiSymbol.Show'}
	{attribute 'TcHmiSymbol.ReadOnly'}
	bAlarm:			BOOL;
	{attribute 'TcHmiSymbol.Show'}
	{attribute 'TcHmiSymbol.ReadOnly'}
	bPressureAlarm:	BOOL := FALSE;
	{attribute 'TcHmiSymbol.Show'}
	{attribute 'TcHmiSymbol.ReadOnly'}
	bPumpAlarm:		BOOL := FALSE;


	// Generic controller OK flag.
	// Used for problems other than from the actuator.
	// This flag is used for problems coming from controllers
	// that extend the functionality of FB_CRYO_BIN_CTRL.
	bCtrlOK:	BOOL := TRUE;		

	nState:			E_NOTT_CRYO_WARMUP_STATE := E_NOTT_CRYO_WARMUP_STATE.NONE;
	
	sErrorText:		STRING(64);		// Error as text
	sState:			STRING(64);		// State as text
	{attribute 'TcHmiSymbol.Show'}
	{attribute 'TcHmiSymbol.ReadOnly'}
	sStatus:		STRING(64);		// Status as text
END_STRUCT
END_TYPE

// ---- POUs/MAIN.TcPOU
PROGRAM MAIN
VAR
		{attribute 'TcHmiSymbol.Show'}
	nott_cryo_ctrl : FB_NOTT_CRYO_CTRL;
END_VAR


nott_cryo_ctrl();

END_PROGRAM

// ---- POUs/FB_NOTT_CRYO_CTRL.TcPOU
// NOTT Cryogenic Controller
FUNCTION_BLOCK FB_NOTT_CRYO_CTRL
VAR_INPUT
	in_sName:	STRING := 'NOTT_CRYO_CTRL';	// Control System name
END_VAR
VAR

	///////////////////////////
	// Configuration parameters
	///////////////////////////
	cfg:	T_NOTT_CRYO_CFG;
	
	/////////////////////
	// Control parameters
	/////////////////////
	{attribute 'TcHmiSymbol.Show'}
	ctrl:	T_NOTT_CRYO_CTRL;

	/////////////////////
	// Status parameters
	/////////////////////
	{attribute 'OPC.UA.DA' := '1'}
	{attribute 'OPC.UA.DA.Access' := '1'}
	{attribute 'TcHmiSymbol.Show'}
	stat:	T_NOTT_CRYO_STAT;

	/////////////////////
	// Debug parameters
	/////////////////////
	debug:	T_NOTT_CRYO_DEBUG;

	/////////////////////
	// System Triggers
	/////////////////////
	triggers:	T_NOTT_CRYO_TRIGGERS;

	/////////////////////
	// System Events
	/////////////////////
	events:	T_NOTT_CRYO_EVENTS;

	/////////////////////
	// Local variables
	/////////////////////
	bCoolDownPermitEvacuationStop:	BOOL := FALSE;
	bCoolDownPermitWarmUp:			BOOL := FALSE;
	bWarmUpPermitEvacuationStop:	BOOL := FALSE;
	bWarmUpPermitCoolDown:			BOOL := FALSE;


	//////////////////////////////////////////////
	//             Controllers
	//////////////////////////////////////////////
 	{attribute 'TcHmiSymbol.Show'}
 	cool_down:			FB_NOTT_CRYO_COOLDOWN;
	{attribute 'TcHmiSymbol.Show'}
 	warm_up:			FB_NOTT_CRYO_WARMUP;

	
	//
	// Heaters
	//
// 	{attribute 'TcHmiSymbol.Show'}
// 	Heater_DetIF:		FB_PDS_CRYO_HEATER_CTRL;
// 	{attribute 'TcHmiSymbol.Show'}
// 	Heater_Preamp:		FB_PDS_CRYO_HEATER_CTRL;
// 	{attribute 'TcHmiSymbol.Show'}
// 	Heater_ColdPlate:	FB_PDS_CRYO_HEATER_CTRL;
// 	
// 	//
// 	// Pointers to System Overrides for control and sensors.
// 	// See M_Configure() for pointer assignments.
// 	//
// 	// Pointers to Overrides of Enable commands for valves, pumps and coolers.
	ptrArr_cor:	ARRAY [0..7] OF POINTER TO FB_CRYO_CMD_OVERRIDE;
	// Pointers to Overrides of Simulation flags for Temperatures.
// 	// Must match indexes of ptrArr_Temp[], see below.
	ptrArr_tor:	ARRAY [0..8] OF POINTER TO FB_CRYO_CMD_OVERRIDE;
// 	// Pointers to Overrides of Simulation flags for Pressures.
	ptrArr_por:	ARRAY [0..1] OF POINTER TO FB_CRYO_CMD_OVERRIDE;
// 	
// 	//
// 	// Indexes for Override GUIs.
// 	//
	guiIndex_cor:	UINT := 0;	// Index for Command Override Engineering GUI
	guiIndex_tor:	UINT := 0;	// Index for Temperature Override Engineering GUI
	guiIndex_por:	UINT := 0;	// Index for Pressure Override Engineering GUI
// 	
// 
	//////////////////////////////////////////////
	//             Subsystems
	//////////////////////////////////////////////

	//
	// Evacuation Subsystem control
	//
	{attribute 'TcHmiSymbol.Show'}
	evac:			FB_NOTT_CRYO_EVAC;	// PDS Evacuation Subsystem
	
	

	//////////////////////////////////////////////
	//             Sensors
	//////////////////////////////////////////////
	// Cryostat Pressure sensors
	sensor_VAGC:	FB_CRYO_SENSOR_PRESSURE;	// Cryo pressure gauge VAGC
	VAGC:			FB_CRYO_PRESSURE_VOTE;		// Cryo pressure C
	
		// Cryostat High Pressure sensor
	sensor_HPG:	FB_CRYO_SENSOR_PRESSURE;	// Cryo pressure gauge VAGC
	HPG:			FB_CRYO_PRESSURE_VOTE;		// Cryo pressure C

	///////////////////////////////////////////////////////
	//                  Temperatures
	///////////////////////////////////////////////////////
 
	{attribute 'OPC.UA.DA' := '1'}
	{attribute 'TcHmiSymbol.Show'}
 	nott_temp:				FB_NOTT_TEMPERATURES;  // All temperature sensors

	
	    /////////////////////////////////////////////////////////
	////                  Voters
	/////////////////////////////////////////////////////////
	{attribute 'OPC.UA.DA' := '1'}
		{attribute 'TcHmiSymbol.Show'}
    nott_voters : FB_NOTT_VOTERS; // All METIS voters

	/////////////////////////////////////////////////////////
	////                  Temperature control
	/////////////////////////////////////////////////////////
	{attribute 'OPC.UA.DA' := '1'}
		{attribute 'TcHmiSymbol.Show'}
// 	nott_tctrl:              FB_NOTT_TCTRL; // All temperature control loops
    
    /////////////////////////////////////////////////////////
	////                  Heaters
	/////////////////////////////////////////////////////////
	{attribute 'OPC.UA.DA' := '1'}
		{attribute 'TcHmiSymbol.Show'}
 	nott_heaters:			FB_NOTT_HEATERS; // All METIS heaters

	/////////////////////////////////////////////////////////
	////                  Temperature control
	/////////////////////////////////////////////////////////
	{attribute 'OPC.UA.DA' := '1'}
		{attribute 'TcHmiSymbol.Show'}
	nott_tctrl:              FB_NOTT_TCTRLs; // All temperature control loops


	/////////////////////////////////////////////////////////
	////                  Thermal Box Control
	/////////////////////////////////////////////////////////
	
	{attribute 'OPC.UA.DA' := '1'}
	{attribute 'TcHmiSymbol.Show'}
	thermal_box_ctrl:	FB_NOTT_THERMAL_BOX_CONTROL; // Fan and water-valve temperature control


	ptrArr_Temp:	ARRAY [0..8] OF POINTER TO FB_CRYO_TEMPERATURE;
// 	// Pointers to Pressures.
	ptrArr_Press:	ARRAY [0..1] OF POINTER TO FB_CRYO_PRESSURE_VOTE;
// 	
// 	//
// 	// System triggers
// 	//	
	{attribute 'OPC.UA.DA' := '0'}
	trgCool:			R_TRIG;
	{attribute 'OPC.UA.DA' := '0'}
	trgCoolStop:		F_TRIG;
	{attribute 'OPC.UA.DA' := '0'}
	trgWarmup:			R_TRIG;
	{attribute 'OPC.UA.DA' := '0'}
	trgWarmupStop:		F_TRIG;
	{attribute 'OPC.UA.DA' := '0'}
	trgEvacOn:			R_TRIG;
	{attribute 'OPC.UA.DA' := '0'}
	trgEvacOff:			F_TRIG;

	{attribute 'OPC.UA.DA' := '0'}
	timer:		TON;		// Timer for commands
	
	
	//
	//	Input signals
	//	
	
	
	//
	// Dummy values for simulation, etc.
	//
	// Dummy OP state for mapping of simulated devices.
	q_nStateDummy	AT%Q*:	UINT := 8;		

// 	// HMI Parameters
	hmi_pump_tmp: FB_HMI_CRYO_PUMP;
	hmi_pump_pvp: FB_HMI_CRYO_PUMP;
	hmi_valve_pvv1: FB_HMI_CRYO_VALVE;
	hmi_cooler: FB_HMI_CRYO_HELIUM_COMPRESSOR;
	
	
// 	hmi_lakeshore : FB_HMI_CRYO_LAKESHORE;
// 	hmi_heater_DetIF : FB_HMI_PDS_CRYO_HEATER;
// 	hmi_heater_Preamp : FB_HMI_PDS_CRYO_HEATER;
// 	hmi_heater_ColdPlate : FB_HMI_PDS_CRYO_HEATER;
	hmi_pressure_vote_vagc : FB_HMI_CRYO_PRESSURE_VOTE;
	hmi_pressure_vote_vag1 : FB_HMI_CRYO_PRESSURE_VOTE;
	hmi_pressure_vote_hpg : FB_HMI_CRYO_PRESSURE_VOTE;
// 
// 	hmi_heater_DetIF_temp : FB_HMI_CRYO_TEMPERATURE;
// 	hmi_heater_Preamp_temp : FB_HMI_CRYO_TEMPERATURE;
// 	hmi_heater_Coldplate_temp : FB_HMI_CRYO_TEMPERATURE;

	// Alarm Handling
	fbEventAlarm    : ARRAY[0..2] OF FB_EventAlarm;
	arrAlarmState    : ARRAY[0..2] OF BOOL;
	
	// Cryo System logs
	logs:	FB_CRYO_FUNCTION_LOG;

	
	////////////////////
	//// HMI Screen /// 
	//////////////////

bHMISwitch     AT %I* : BOOL;   // Push button / switch
bHMIOutEnable  AT %Q* : BOOL;   // HMI power output;

END_VAR

// Increment cycle counter
debug.nCycleCounter := debug.nCycleCounter + 1;

//Wait UNTIL the controller is configured.
IF NOT stat.bConfigured THEN
	M_Configure(); 
	RETURN;
END_IF


//
// Read Temperature and Pressure Sensors

M_ReadSensors();


//
// Check for sensor HW errors
//
// M_CheckForSensorErrors();



///////////////////
// System Operation
///////////////////

//
// Execute Controllers
//
M_ExecuteControllers();


//
// Update command permissions
//
M_SetCmdPermissions();


//
// Capture system commands
//
M_CheckForCommands();


//
// Perform a safety check
//
M_SafetyCheck();


//
// Check triggers and log events
//
M_ProcessTriggers();

M_ProcessHmi();

//
// Execute system state machine
//
M_StateMachine();

//
// Refresh permissions after state transitions
//
M_SetCmdPermissions();

//
// HMI Screen ON/OFF
//
M_HMI_Screen_Control();

METHOD M_CheckForCommands
VAR_INPUT
END_VAR


// Capture Cooldown ON/OFF command
trgCool(CLK := ctrl.bEnable_CoolDown);
trgCoolStop(CLK := ctrl.bEnable_CoolDown);

IF trgCool.Q THEN
	IF cool_down.bPermitStart THEN
		ctrl.bExecute	:= TRUE;
		ctrl.nCommand	:= E_NOTT_CRYO_CTRL_CMD.COOL;
	ELSE
		ctrl.bEnable_CoolDown	:= FALSE;
		logs.M_LogInfo('Cooldown start command rejected: permission denied.');
	END_IF

ELSIF trgCoolStop.Q THEN
	IF cool_down.bPermitStop THEN
		logs.M_LogInfo('Cooldown stop command accepted.');
	ELSE
		// Do not force ctrl.bEnable_CoolDown back to TRUE here.
		// The state machine also writes this bit internally.
		logs.M_LogInfo('Cooldown stop command not permitted.');
	END_IF
END_IF

// Capture Evacuation ON/OFF trigger
trgEvacOn(CLK := ctrl.bEnable_Evac);
trgEvacOff(CLK := ctrl.bEnable_Evac);

IF trgEvacOn.Q THEN
	IF evac.bPermitStart THEN
		ctrl.bEnable_Evac := TRUE;
		logs.M_LogInfo('Evacuation started.');
	ELSE
		ctrl.bEnable_Evac := FALSE;
		logs.M_LogInfo('Evacuation start command rejected: permission denied.');
	END_IF

ELSIF trgEvacOff.Q THEN
	IF evac.bPermitStop THEN
		ctrl.bEnable_Evac := FALSE;
		logs.M_LogInfo('Evacuation stopped.');
	ELSE
		// Do not force ctrl.bEnable_Evac back to TRUE here.
		logs.M_LogInfo('Evacuation stop command not permitted.');
	END_IF
END_IF


// Capture Evacuation ON/OFF trigger
trgEvacOn(CLK := ctrl.bEnable_Evac);
trgEvacOff(CLK := ctrl.bEnable_Evac);

IF trgEvacOn.Q THEN
	IF evac.bPermitStart THEN
		ctrl.bEnable_Evac := TRUE;
		logs.M_LogInfo('Evacuation started.');
	ELSE
		ctrl.bEnable_Evac := FALSE;
		logs.M_LogInfo('Evacuation start command rejected: permission denied.');
	END_IF

ELSIF trgEvacOff.Q THEN
	IF evac.bPermitStop THEN
		ctrl.bEnable_Evac := FALSE;
		logs.M_LogInfo('Evacuation stopped.');
	ELSE
		// Do not force ctrl.bEnable_Evac back to TRUE here.
		logs.M_LogInfo('Evacuation stop command not permitted.');
	END_IF
END_IF
END_METHOD

METHOD M_CheckForSensorErrors
VAR_INPUT
END_VAR
// Don't do any checks on startup.

IF stat.nState = E_NOTT_CRYO_CTRL_STATE.NONE	THEN
	RETURN;
END_IF


////////////////////////////////////////////////
// Check for errors by testing the 'Valid' flag.
////////////////////////////////////////////////
IF	NOT VAGC.stat.bValid	THEN
	stat.bError	:= TRUE;
	stat.sState	:= 'Cryo Vacuum gauge problem';
	IF stat.nState	<> E_NOTT_CRYO_CTRL_STATE.ERROR	THEN
		logs.M_LogInfo('ERROR State: VAGC gauge failure');
	END_IF
	stat.nState	:= E_NOTT_CRYO_CTRL_STATE.ERROR;

ELSE
	stat.bError	:= FALSE;
//	stat.sState	:= '';
END_IF


///////////////////////
// Check for Interlocks
///////////////////////
// TODO

//
// Evacuation and Repressurization are mutually exclusive.
//
// TODO


//
// Disable control in failure state
//
IF stat.bError THEN
	ctrl.bEnable_CoolDown 	:= FALSE;
	ctrl.bEnable_Warmup		:= FALSE;
END_IF
END_METHOD

METHOD M_CheckLakeshoreCommand
VAR_INPUT
END_VAR
(* TODO

IF ctrl.bLS_UpdateSETP THEN
Reset trigger flag
	ctrl.bLS_UpdateSETP	:= FALSE;
	
Safety
	IF ctrl.lrLS_RAMP > 1.0 THEN
		ctrl.lrLS_RAMP	:= 1.0;
	ELSIF ctrl.lrLS_RAMP < 0.0 THEN
		ctrl.lrLS_RAMP	:= 0.0;
	END_IF
	
Set the mode
	IF ctrl.nLS_Mode <> E_CRYO_LAKESHORE_MODE.MONITORING THEN
		Lakeshore.M_SetMode(ctrl.nLS_Mode);
	ELSE
		RETURN;	// Nothing to do
	END_IF
ELSE
	RETURN;	// Nothing to do
END_IF




CASE ctrl.nLS_Mode OF
	E_CRYO_LAKESHORE_MODE.MONITORING,
	E_CRYO_LAKESHORE_MODE.COOLING,
	E_CRYO_LAKESHORE_MODE.WARMUP,
	E_CRYO_LAKESHORE_MODE.COOLING_UPDATE,
	E_CRYO_LAKESHORE_MODE.WARMUP_UPDATE:
		Lakeshore.M_SetMode(E_CRYO_LAKESHORE_MODE.MONITORING);	// No action
		
	E_CRYO_LAKESHORE_MODE.SINGLE_SETUP:
		IF stat.nState = E_CRYO_CTRL_STATE.COLD THEN
			Lakeshore.M_SetParams(
				in_nPID_A_P			:= cfg.LS_W_PID_A_P, 
				in_nPID_A_I			:= cfg.LS_W_PID_A_I, 
				in_nPID_A_D			:= cfg.LS_W_PID_A_D, 
				in_nHeater_Range	:= cfg.LS_W_Heater_Range, 
				in_lrCtrlRamp		:= ctrl.lrLS_RAMP, 
				in_lrSetpoint_A		:= ctrl.lrLS_SETP);
		END_IF
	ELSE
		Lakeshore.M_SetMode(E_CRYO_LAKESHORE_MODE.MONITORING);	// No action
END_CASE
*)
END_METHOD

// Method to check status of the cryostat vacuum.
// TODO: The limits might depend on the temperature.
METHOD M_CheckVacuum
VAR_INPUT
END_VAR
VAR_INST
	tonVacuumEntry:		TON;
	tonVacuumExit:		TON;
	tonGoodVacuumEntry:	TON;
	tonGoodVacuumExit:	TON;
END_VAR
VAR CONSTANT
	tVacuumConfirm:	TIME := T#5S;
END_VAR
IF VAGC.stat.bValid THEN
	stat.bPressureValid := TRUE;
	stat.lrPressure_mbar := VAGC.stat.lrPressure;

	// In-vacuum status: enter below 1.0 mbar and leave above 1.2 mbar.
	IF stat.bVacuum THEN
		tonVacuumEntry(IN := FALSE, PT := tVacuumConfirm);
		tonVacuumExit(
			IN := VAGC.stat.lrPressure > cfg.lrPress_InVac_Reset,
			PT := tVacuumConfirm);

		IF tonVacuumExit.Q THEN
			stat.bVacuum := FALSE;
			tonVacuumExit(IN := FALSE, PT := tVacuumConfirm);
		END_IF
	ELSE
		tonVacuumExit(IN := FALSE, PT := tVacuumConfirm);
		tonVacuumEntry(
			IN := VAGC.stat.lrPressure < cfg.lrPress_InVac,
			PT := tVacuumConfirm);

		IF tonVacuumEntry.Q THEN
			stat.bVacuum := TRUE;
			tonVacuumEntry(IN := FALSE, PT := tVacuumConfirm);
		END_IF
	END_IF

	// Good-vacuum status: enter below 0.001 mbar and leave above 0.002 mbar.
	IF stat.bVacuumOK THEN
		tonGoodVacuumEntry(IN := FALSE, PT := tVacuumConfirm);
		tonGoodVacuumExit(
			IN := VAGC.stat.lrPressure > cfg.lrPress_GoodVac_Reset,
			PT := tVacuumConfirm);

		IF tonGoodVacuumExit.Q THEN
			stat.bVacuumOK := FALSE;
			tonGoodVacuumExit(IN := FALSE, PT := tVacuumConfirm);
		END_IF
	ELSE
		tonGoodVacuumExit(IN := FALSE, PT := tVacuumConfirm);
		tonGoodVacuumEntry(
			IN := VAGC.stat.lrPressure < cfg.lrPress_GoodVac,
			PT := tVacuumConfirm);

		IF tonGoodVacuumEntry.Q THEN
			stat.bVacuumOK := TRUE;
			stat.bVacuum   := TRUE;
			tonGoodVacuumEntry(IN := FALSE, PT := tVacuumConfirm);
		END_IF
	END_IF

	// Good vacuum is always a subset of in-vacuum.
	IF stat.bVacuumOK THEN
		stat.bVacuum := TRUE;
	END_IF
ELSE
	stat.bPressureValid := FALSE;
	stat.bVacuum        := FALSE;
	stat.bVacuumOK      := FALSE;

	tonVacuumEntry(IN := FALSE, PT := tVacuumConfirm);
	tonVacuumExit(IN := FALSE, PT := tVacuumConfirm);
	tonGoodVacuumEntry(IN := FALSE, PT := tVacuumConfirm);
	tonGoodVacuumExit(IN := FALSE, PT := tVacuumConfirm);
END_IF
END_METHOD

METHOD M_Configure
VAR_INPUT
END_VAR
VAR
	refBOOL:	REFERENCE TO BOOL;
END_VAR
IF stat.bConfigured THEN
	RETURN;
ELSIF debug.nCycleCounter = 1 THEN
// THIS call just configures logs AT the very start.
// Logging is done by explicit calls to M_LogInfo().
	logs(in_sName := in_sName);
	

	// Set pointers to Pressure readings
	ptrArr_Press[0] := ADR(VAGC);	
	ptrArr_Press[1] := ADR(evac.VAG1);	

	
// Set pointers to Overrides of Simulation flags for Pressures.
	ptrArr_por[0] := ADR(ctrl.por_VAGC);
	ptrArr_por[1] := ADR(evac.ctrl.por_VAG1);
	
ELSIF debug.nCycleCounter = 2 THEN
// Initialize events
	events.info.CreateEx		(TC_EVENTS.NottCryoSysEventClass.Info,0);
	events.warning.CreateEx		(TC_EVENTS.NottCryoSysEventClass.Warning,0);
	events.error.CreateEx		(TC_EVENTS.NottCryoSysEventClass.Error,FALSE,0);
	events.critical.CreateEx	(TC_EVENTS.NottCryoSysEventClass.Critical,TRUE,0);
	
ELSIF debug.nCycleCounter = 3 THEN
	
	
// Pressure Simulation flags
	ctrl.bSim_Press_VAGC		:= FALSE;	// The values will come from the simulator.
	//evac.ctrl.bSim_Press_VAG1	:= FALSE;	// The values will come from the simulator.
	//refBOOL	REF=evac.ctrl.bSim_Press_VAG1;	refBOOL	:= TRUE;

ELSIF debug.nCycleCounter > 200 THEN
	stat.bConfigured	:= TRUE;
ELSE
	RETURN;
END_IF
END_METHOD

METHOD M_ExecuteControllers
VAR
	ptrSimTemp:	POINTER TO LREAL;
END_VAR

nott_tctrl(temperatures := nott_temp);

nott_heaters(tctrl := nott_tctrl);

thermal_box_ctrl(	nott_temps:= nott_temp, 
	nott_heaters:= nott_heaters, 
	nott_t_ctrls:= nott_tctrl, 
	nott_t_votes:= nott_voters);


// //
// // Controllers, i.e. LN2 cooler, Heater, ...
// //
// 
// // Evacuation subsystem
ctrl.cor_Evac(in_bEnable:=ctrl.bEnable_Evac);
evac(	in_bEnable	:= ctrl.cor_Evac.out_bEnable, 
		in_RefVAGC	:= VAGC);	
		
//
// Pump State
//
M_GetPumpsStates();

ctrl.cor_CoolDown(in_bEnable:=ctrl.bEnable_CoolDown);
cool_down(
	in_bEnable:= ctrl.cor_CoolDown.out_bEnable,
	in_Cryo_Stat := stat, 
	out_bPermit_Evacuation_Stop=> bCoolDownPermitEvacuationStop, 
	out_bPermit_WarmUp=> bCoolDownPermitWarmUp, 
	nott_temps:= nott_temp, 
	nott_heaters:= nott_heaters, 
	nott_t_ctrls:= nott_tctrl, 
	nott_t_votes:= nott_voters);

ctrl.cor_WarmUp(in_bEnable:=ctrl.bEnable_WarmUp);
warm_up(
	in_bEnable:= ctrl.cor_WarmUp.out_bEnable,
	in_Cryo_Stat := stat, 
	out_bPermit_Evacuation_Stop=> bWarmUpPermitEvacuationStop, 
	out_bPermit_CoolDown=> bWarmUpPermitCoolDown, 
	nott_temps:= nott_temp, 
	nott_heaters:= nott_heaters, 
	nott_t_ctrls:= nott_tctrl, 
	nott_t_votes:= nott_voters);


// Update the combined thermal and operational status flags.
M_UpdateThermalStatus();


//
// Get the lowest temperature in the cryostat
//	
M_GetLowestTemperature();

//
// Get the highest temperature in the cryostat
//	
M_GetHighestTemperature();
END_METHOD

METHOD M_GetHighestTemperature
VAR_INPUT
END_VAR
VAR
	lrTempK:	LREAL	:= 0.0;	// The lowest possible temperature
	bValid:		BOOL	:= FALSE;
	i:			INT;
END_VAR


stat.lrHighestTempK		:= nott_temp.out_lrHighestTemp;
stat.bHighestTempValid	:= nott_temp.out_bHighestTempValid;
stat.sHighestTempName	:= nott_temp.out_sHighestTempName;
END_METHOD

METHOD M_GetLowestTemperature
VAR_INPUT
END_VAR
VAR
	lrTempK:	LREAL	:= 850.0;	// Highest possible temperature
	bValid:		BOOL	:= FALSE;
	i:			INT;
END_VAR


stat.lrLowestTempK		:= nott_temp.out_lrLowestTemp;
stat.bLowestTempValid	:= nott_temp.out_bLowestTempValid;
stat.sLowestTempName	:= nott_temp.out_sLowestTempName;
END_METHOD

METHOD M_GetPumpsStates : BOOL
VAR_INPUT
END_VAR
// Pump ready/failure flags are not populated reliably. Use the real-time
// monitored speeds as the authoritative running indications.
stat.bIsPVPRunning := evac.pump_pvp.stat.nPumpSpeed > 10;
stat.bIsTMPRunning := evac.pump_tmp.stat.nPumpSpeed > 10;

M_GetPumpsStates := stat.bIsPVPRunning AND stat.bIsTMPRunning;
END_METHOD

METHOD M_GetState
VAR_INPUT
END_VAR
VAR_INST
	timer:		TON;
END_VAR
// Determine the initial state based on the command and actuator state.

// Firstly wait for the complete system to start.
// Serial port devices need about seven seconds to initialise.
// We wait 10 sec to avoid going into Error state on startup.
//
IF NOT stat.bSystemStarted	THEN
	// Start the 10s timer
	timer(IN:=FALSE);
	timer(IN:=TRUE, PT:=T#10S);
	stat.bSystemStarted	:= TRUE;
	stat.sState	:= 'Starting...';
	RETURN;
END_IF

timer();

IF timer.Q	OR stat.bSystemStarted THEN
	timer(IN:=FALSE);	// Reset the timer
	
	// 10S have expired.
	// Find the system state from the combined thermal and pressure statuses.
	// If temperature or pressure status cannot be estimated, the logic falls
	// through to WARM_PRESS as the conservative startup state.
	IF stat.bOP OR stat.bCold	THEN
		logs.M_LogInfo('On restart, System is COLD.');
		// Turn ON the Cool-Down 
		ctrl.bEnable_CoolDown	:= TRUE;
		// Enable Evacuation
		ctrl.bEnable_Evac	:= TRUE;
		//Disable WarmUp
		ctrl.bEnable_WarmUp := FALSE;
		// Log
		logs.M_LogInfo('System started in state COLD');
		// Switch to Cold state.
		stat.nState	:= E_NOTT_CRYO_CTRL_STATE.COLD;
		
	ELSIF stat.bVacuumOK OR stat.bVacuum THEN
		// Enable Evacuation
		ctrl.bEnable_Evac		:= TRUE;
		// Stop Cooler.
		ctrl.bEnable_CoolDown	:= FALSE;
		// Turn OFF the heaters.
		ctrl.bEnable_WarmUp	:= FALSE;
		// Log
		logs.M_LogInfo('System started in state WARM_VACUUM');

		// The system is in WARM_VACUUM.
		stat.nState := E_NOTT_CRYO_CTRL_STATE.WARM_VACUUM;		
		
	ELSE
		// Stop Evacuation.
		ctrl.bEnable_Evac			:= FALSE;
		// Stop Cooler.
		ctrl.bEnable_CoolDown		:= FALSE;
		// Turn OFF the heaters.
		ctrl.bEnable_WarmUp			:= FALSE;
		logs.M_LogInfo('System started in state WARM_PRESS');

		// The system is in WARM_PRESS.
		stat.nState := E_NOTT_CRYO_CTRL_STATE.WARM_PRESS;
	END_IF	
ELSE
	stat.sState	:= 'Starting...';
END_IF

// // Determine the initial state based on the command and actuator state.
// 
// // Firstly wait for the complete system to start.
// // Serial port devices need about seven seconds to initialise.
// // We wait 10 sec to avoid going into Error state on startup.
// //
// IF NOT stat.bSystemStarted	THEN
// 	// Start the 10s timer
// 	timer(IN:=FALSE);
// 	timer(IN:=TRUE, PT:=T#10S);
// 	stat.bSystemStarted	:= TRUE;
// 	stat.sState	:= 'Starting...';
// 	RETURN;
// END_IF
// 
// timer();
// 
// IF timer.Q	THEN
// 	timer(IN:=FALSE);	// Reset the timer
// 	
// 	// 10S have expired.
// 	// Find the system state based of sensor eadings.
// 	IF nott_voters.vote_detector.stat.lrTempK < cfg.lrTemp_Warm	THEN
// 		logs.M_LogInfo('On restart, System is COLD.');
// 		// Turn ON the Cool-Down 
// 		ctrl.bEnable_CoolDown	:= TRUE;
// 		// Enable Evacuation
// 		ctrl.bEnable_Evac	:= TRUE;
// 		//Disable WarmUp
// 		ctrl.bEnable_WarmUp := FALSE;
// 		// Log
// 		logs.M_LogInfo('System started in state COLD');
// 		// Switch to Cold state.
// 		stat.nState	:= E_NOTT_CRYO_CTRL_STATE.COLD;
// 		
// 	ELSIF 	nott_voters.vote_detector.stat.lrTempK >= cfg.lrTemp_Warm	AND 
// 			VAGC.stat.lrPressure <= cfg.lrPress_InVac				THEN
// 		// Enable Evacuation
// 		ctrl.bEnable_Evac		:= TRUE;
// 		// Stop Cooler.
// 		ctrl.bEnable_CoolDown	:= FALSE;
// 		// Turn OFF the heaters.
// 		ctrl.bEnable_WarmUp	:= FALSE;
// 		// Log
// 		logs.M_LogInfo('System started in state WARM_VACUUM');
// 
// 		// The system is in WARM_VACUUM.
// 		stat.nState := E_NOTT_CRYO_CTRL_STATE.WARM_VACUUM;		
// 		
// 	ELSIF 	nott_voters.vote_detector.stat.lrTempK >= cfg.lrTemp_Warm	AND 
// 			VAGC.stat.lrPressure > cfg.lrPress_InVac				THEN
// 		// Stop Evacuation.
// 		ctrl.bEnable_Evac	:= FALSE;
// 		// Stop Cooler.
// 		ctrl.bEnable_CoolDown		:= FALSE;
// 		// Turn OFF the heaters.
// 		ctrl.bEnable_WarmUp	:= FALSE;
// 		logs.M_LogInfo('System started in state WARM_PRESS');
// 
// 		// The system is in WARM_PRESS.
// 		stat.nState := E_NOTT_CRYO_CTRL_STATE.WARM_PRESS;
// 	ELSE
// // Stop Evacuation.
// 		ctrl.bEnable_Evac			:= FALSE;
// // Stop Cooler.
// 		ctrl.bEnable_CoolDown		:= FALSE;
// // Turn OFF the heaters.
// 		ctrl.bEnable_WarmUp			:= FALSE;
// 		logs.M_LogInfo('System started in state WARM_PRESS');
// 
// // The system is in WARM_PRESS.
// 		stat.nState := E_NOTT_CRYO_CTRL_STATE.WARM_PRESS;
// 	END_IF	
// ELSE
// 	stat.sState	:= 'Starting...';
// END_IF
END_METHOD

METHOD M_HMI_Screen_Control : BOOL
VAR_INPUT
END_VAR
VAR_INST
    trigHMISwitch : R_TRIG;
END_VAR
M_HMI_Screen_Control := TRUE;

////////////////////
/// HMI Screen   ///
////////////////////

// Rising edge detection
trigHMISwitch(CLK := bHMISwitch);

// Toggle HMI power output
IF trigHMISwitch.Q THEN
    bHMIOutEnable := NOT bHMIOutEnable;
END_IF
END_METHOD

METHOD PRIVATE M_ProcessHmi
hmi_pump_tmp(
	inout_sPumpStatRef := evac.pump_tmp.stat,
	inout_sCmdOver := evac.ctrl.cor_TMP,
	inout_fbAlarmHandlerRef := evac.pump_tmp.fbAlarmHandler
	);

hmi_pump_pvp(
	inout_sPumpStatRef := evac.pump_pvp.stat,
	inout_sCmdOver := evac.ctrl.cor_PVP,
	inout_fbAlarmHandlerRef := evac.pump_pvp.fbAlarmHandler
	);

hmi_valve_pvv1(
	inout_sValveStatRef := evac.PVV1.stat,
	inout_sCmdOver := evac.ctrl.cor_PVV1,
	inout_fbAlarmHandlerRef := evac.PVV1.fbAlarmHandler,
	);
	
hmi_cooler(inout_sCpaStatRef:= cool_down.cooler.stat, inout_sCmdOver:= cool_down.ctrl.cor_Cooler, out_stat=> );


hmi_pressure_vote_vagc(
	inout_sPressureVoteStatRef := VAGC.stat,
	inout_sCmdOver := ctrl.por_VAGC,
	inout_fbAlarmHandlerRef := VAGC.fbAlarmHandler
	);

hmi_pressure_vote_vag1(
	inout_sPressureVoteStatRef := evac.VAG1.stat,
	inout_sCmdOver := evac.ctrl.por_VAG1,
	inout_fbAlarmHandlerRef := evac.VAG1.fbAlarmHandler
	);
hmi_pressure_vote_hpg(
	inout_sPressureVoteStatRef := HPG.stat,
	inout_sCmdOver := ctrl.por_HPG,
	inout_fbAlarmHandlerRef := HPG.fbAlarmHandler
	);
END_METHOD

METHOD M_ProcessTriggers
VAR_INPUT
END_VAR
VAR
    fbFormat:	FB_FormatString;
	sOut:		STRING;
END_VAR
//
// Check triggers and log corresponding events.
//

//
// Cooler
//
// triggers.Cooler_Enable		(CLK := cooler.in_bEnable);
// triggers.Cooler_Disable		(CLK := cooler.in_bEnable);
// triggers.Cooler_ON			(CLK := (cooler.stat.nDevState = E_CRYO_CRYOTELGT_STATE.ON));
// triggers.Cooler_OFF			(CLK := (cooler.stat.nDevState = E_CRYO_CRYOTELGT_STATE.OFF));
// 
// IF triggers.Cooler_Enable.Q	THEN
// 	logs.M_LogInfo('Cooler Starting...');
// ELSIF triggers.Cooler_Disable.Q	THEN
// 	logs.M_LogInfo('Cooler Stopping...');
// ELSIF triggers.Cooler_ON.Q	THEN
// 	logs.M_LogInfo('Cooler ON');
// ELSIF triggers.Cooler_OFF.Q	THEN
// 	logs.M_LogInfo('Cooler OFF');
// END_IF


//
// Pressure and Temperature status flags
//

// Vacuum
triggers.Vacuum_ON		(CLK := stat.bVacuum);
triggers.Vacuum_OFF		(CLK := stat.bVacuum);
triggers.Vacuum_OK		(CLK := stat.bVacuumOK);
triggers.Vacuum_NOT_OK	(CLK := stat.bVacuumOK);

IF triggers.Vacuum_ON.Q	THEN
	logs.M_LogInfo('In Vacuum');
ELSIF triggers.Vacuum_OFF.Q	THEN
	logs.M_LogInfo('NOT In Vacuum');
ELSIF triggers.Vacuum_OK.Q	THEN
	logs.M_LogInfo('Vacuum OK');
ELSIF triggers.Vacuum_NOT_OK.Q	THEN
	logs.M_LogInfo('Vacuum NOT OK');
END_IF


// Temperature
triggers.Cold_ON		(CLK := stat.bCold);
triggers.Cold_OFF		(CLK := stat.bCold);
triggers.OP_ON			(CLK := stat.bOP);
triggers.OP_OFF			(CLK := stat.bOP);

IF triggers.Cold_ON.Q	THEN
	logs.M_LogInfo('System is COLD');
ELSIF triggers.Cold_OFF.Q	THEN
	logs.M_LogInfo('System is NOT COLD');
ELSIF triggers.OP_ON.Q	THEN
	logs.M_LogInfo('System is OPERATIONAL');
ELSIF triggers.OP_OFF.Q	THEN
	logs.M_LogInfo('System is NOT OPERATIONAL');
END_IF
END_METHOD

METHOD M_ReadSensors
VAR_INPUT
END_VAR
VAR
	refBOOL:	REFERENCE TO BOOL;
	refLREAL:	REFERENCE TO LREAL;
END_VAR
//
// Read system temperatures.
//

nott_temp();

// Update the voters
nott_voters(nott_temp := nott_temp);


// NOTT Cryostat pressure.

// Sensor instance
// Average over 1 sec (1000 ms).
sensor_VAGC(
	in_sName := 'VAGC_S1',
	in_nType		:= E_CRYO_SENSOR_TYPE_PRESS.PKR_360,	
	in_nSampleTime	:= 1000);

// VAGC Pressure Voting system (one sensor only!)
ctrl.por_VAGC(in_bEnable := ctrl.bSim_Press_VAGC);
VAGC(
	in_sName := 'VAGC',
	in_bSimulation	:= ctrl.por_VAGC.out_bEnable,
// In reality, there is only one pressure sensor connected (sensor_VAGC)
	in_nNumSensor	:= 2,	
	in_nVoteMethod	:= E_CRYO_VOTE.V_1oo2,
	in_pSensor1		:= ADR(sensor_VAGC));
	
sensor_HPG(
	in_sName := 'HPG_S1',
	in_nType		:= E_CRYO_SENSOR_TYPE_PRESS.CMR_361,	
	in_nSampleTime	:= 1000);

//VAGC Pressure Voting system (one sensor only!)
ctrl.por_HPG(in_bEnable := ctrl.bSim_Press_HPG);
HPG(
	in_sName := 'HPG',
	in_bSimulation	:= ctrl.por_HPG.out_bEnable,
// In reality, there is only one pressure sensor connected (sensor_VAGC)
	in_nNumSensor	:= 2,	
	in_nVoteMethod	:= E_CRYO_VOTE.V_1oo2,
	in_pSensor1		:= ADR(sensor_HPG));


//
// Check Vacuum in the system
//	
M_CheckVacuum();
END_METHOD

METHOD M_SafetyCheck
VAR_INPUT
END_VAR
// A pump trip stops the active thermal routine. The routine safety methods
// already disable their actuators and latch the detailed pump alarm.
IF cool_down.stat.bPumpAlarm THEN
	ctrl.bEnable_CoolDown := FALSE;
END_IF

IF warm_up.stat.bPumpAlarm THEN
	ctrl.bEnable_WarmUp := FALSE;
END_IF
END_METHOD

METHOD M_SetCmdPermissions : BOOL
VAR_INPUT
END_VAR
VAR
	bPermitStartEvacuation:	BOOL := FALSE;
	bPermitStopEvacuation:	BOOL := FALSE;
	bPermitStartCoolDown:	BOOL := FALSE;
	bPermitStopCoolDown:	BOOL := FALSE;
	bPermitStartWarmUp:	BOOL := FALSE;
	bPermitStopWarmUp:	BOOL := FALSE;
	bPumpsRunning:		BOOL := FALSE;
END_VAR
M_SetCmdPermissions := FALSE;

bPumpsRunning := stat.bIsPVPRunning AND stat.bIsTMPRunning;

// Start from a fail-closed permission set. Then open the allowed HMI
// actions according to the top-level physical state and active routine.
IF warm_up.stat.bActive THEN
	// Warmup active
	bPermitStartEvacuation	:= TRUE;
	bPermitStopEvacuation	:= FALSE;
	bPermitStartCoolDown	:= FALSE;
	bPermitStopCoolDown		:= FALSE;
	bPermitStartWarmUp		:= TRUE;
	bPermitStopWarmUp		:= TRUE;

ELSIF cool_down.stat.bActive THEN
	// Cooldown active
	bPermitStartEvacuation	:= TRUE;
	bPermitStopEvacuation	:= bCoolDownPermitEvacuationStop AND stat.bOP;
	bPermitStartCoolDown	:= TRUE;
	bPermitStopCoolDown		:= TRUE;
	bPermitStartWarmUp		:= FALSE;
	bPermitStopWarmUp		:= FALSE;

ELSIF stat.bOP THEN
	// Operational
	bPermitStartEvacuation	:= TRUE;
	bPermitStopEvacuation	:= TRUE;
	bPermitStartCoolDown	:= TRUE;
	bPermitStopCoolDown		:= TRUE;
	bPermitStartWarmUp		:= TRUE;
	bPermitStopWarmUp		:= TRUE;

// ELSIF stat.bCold THEN
// 	// Cold but not operational
// 	bPermitStartEvacuation	:= TRUE;
// 	bPermitStopEvacuation	:= FALSE;
// 	bPermitStartCoolDown	:= TRUE;
// 	bPermitStopCoolDown		:= TRUE;
// 	bPermitStartWarmUp		:= FALSE;
// 	bPermitStopWarmUp		:= FALSE;

ELSIF stat.bCold THEN
    // Cold but not operational
    bPermitStartEvacuation := TRUE;
    bPermitStopEvacuation  := FALSE;
    bPermitStartCoolDown   := TRUE;
    bPermitStopCoolDown    := TRUE;
    bPermitStartWarmUp     := TRUE;  // Change from FALSE
    bPermitStopWarmUp      := FALSE;

ELSIF evac.bEvacuationActive THEN
	// Evacuating
	bPermitStartEvacuation	:= TRUE;
	bPermitStopEvacuation	:= TRUE;
	bPermitStartCoolDown	:= TRUE;
	bPermitStopCoolDown		:= FALSE;
	bPermitStartWarmUp		:= FALSE;
	bPermitStopWarmUp		:= FALSE;

ELSIF stat.bVacuumOK OR stat.bVacuum THEN
	// Warm vacuum or good vacuum
	bPermitStartEvacuation	:= TRUE;
	bPermitStopEvacuation	:= TRUE;
	bPermitStartCoolDown	:= TRUE;
	bPermitStopCoolDown		:= FALSE;
	bPermitStartWarmUp		:= FALSE;
	bPermitStopWarmUp		:= FALSE;

ELSE
	// Warm pressurized
	bPermitStartEvacuation	:= TRUE;
	bPermitStopEvacuation	:= FALSE;
	bPermitStartCoolDown	:= FALSE;
	bPermitStopCoolDown		:= FALSE;
	bPermitStartWarmUp		:= FALSE;
	bPermitStopWarmUp		:= FALSE;
END_IF

// Cross-routine vetoes. The routine-specific state machines know when a
// dependent command is safe from their local process state.
bPermitStopEvacuation	:= bPermitStopEvacuation
	AND bCoolDownPermitEvacuationStop
	AND bWarmUpPermitEvacuationStop;

// Evacuation being active does not mean that vacuum has been achieved.
// Apply the physical pressure condition as a final veto to every permission
// branch. stat.bVacuum already includes pressure validity, hysteresis and the
// configured confirmation time from M_CheckVacuum().


bPermitStartCoolDown :=
    bPermitStartCoolDown
    AND bWarmUpPermitCoolDown
    AND stat.bPressureValid
    AND stat.bVacuum
    AND (bPumpsRunning OR stat.bOP);
	
bPermitStartWarmUp		:= bPermitStartWarmUp
	AND bCoolDownPermitWarmUp
	AND bPumpsRunning;

evac.M_PermitStart_Evacuation(in_bPermissionStart := bPermitStartEvacuation);
evac.M_PermitStop_Evacuation(in_bPermissionStop := bPermitStopEvacuation);

cool_down.M_PermitStart_Cooldown(in_bPermissionStart := bPermitStartCoolDown);
cool_down.M_PermitStop_Cooldown(in_bPermissionStop := bPermitStopCoolDown);

warm_up.M_PermitStart_WarmUp(in_bPermissionStart := bPermitStartWarmUp);
warm_up.M_PermitStop_WarmUp(in_bPermissionStop := bPermitStopWarmUp);

ctrl.bSafe_Cooling	:= bPermitStartCoolDown;
ctrl.bSafe_Warmup	:= bPermitStartWarmUp;

M_SetCmdPermissions := TRUE;
END_METHOD

METHOD M_SetStatus
VAR_INPUT
	nState:	E_NOTT_CRYO_CTRL_STATE;
END_VAR

CASE nState OF
	
	E_NOTT_CRYO_CTRL_STATE.NONE:
	stat.bDone	:= TRUE;
	stat.bBusy	:= FALSE;
	stat.bError	:= FALSE;
	stat.bActive:= FALSE;
	stat.sState	:= 'OFF';
	
	E_NOTT_CRYO_CTRL_STATE.WARM_PRESS:
	stat.bDone	:= TRUE;
	stat.bBusy	:= FALSE;
	stat.bError	:= FALSE;
	stat.bActive:= TRUE;
	stat.sState	:= 'WARM - PRESSURIZED';
	
	E_NOTT_CRYO_CTRL_STATE.WARM_VACUUM:
	stat.bDone	:= TRUE;
	stat.bBusy	:= FALSE;
	stat.bError	:= FALSE;
	stat.bActive:= TRUE;
	stat.sState	:= 'WARM - VACUUM';
	

	E_NOTT_CRYO_CTRL_STATE.COOLING_DOWN:
	stat.bDone	:= FALSE;
	stat.bBusy	:= TRUE;
	stat.bError	:= FALSE;
	stat.bActive:= TRUE;
	stat.sState	:= 'COOLING DOWN...';

	E_NOTT_CRYO_CTRL_STATE.COLD:
	stat.bDone	:= TRUE;
	stat.bBusy	:= FALSE;
	stat.bError	:= FALSE;
	stat.bActive:= TRUE;
	stat.sState	:= 'COLD';

	E_NOTT_CRYO_CTRL_STATE.WARMING_UP:
	stat.bDone	:= FALSE;
	stat.bBusy	:= TRUE;
	stat.bError	:= FALSE;
	stat.bActive:= TRUE;
	stat.sState	:= 'WARMING UP...';
	
	// TODO
	// Select reference temperature for warmup
	//
	(*
	IF Temp_Mirror.stat.lrTempK >= cfg.lrTemp_Warm	THEN
		stat.sState	:= 'WARM';
	ELSIF	Temp_Mirror.stat.lrTempK < cfg.lrTemp_Warm AND
			Temp_Mirror.stat.lrTempK >= cfg.lrTemp_Precooled	THEN
		stat.sState	:= 'WARMING UP... PRE-COOLED';
	ELSE
		stat.sState	:= 'WARMING UP... COLD';
	END_IF
	*)

	
	E_NOTT_CRYO_CTRL_STATE.ERROR:
	stat.bDone	:= TRUE;
	stat.bBusy	:= FALSE;
	stat.bError	:= TRUE;
	stat.bActive:= FALSE;
	stat.sState	:= 'ERROR';

END_CASE
END_METHOD

METHOD M_SIM_Cooler
VAR_INPUT
END_VAR
VAR
	refCoolerStat:	REFERENCE TO T_CRYO_CRYOTELGT_STAT;
END_VAR
// // Simulated values
// refCoolerStat	REF=cooler.stat;
// refCoolerStat.nErrorCode	:= 0;
// refCoolerStat.lrTempReject	:= 21.4;
// // Simulated temperature close to DET I/F temperature.
// refCoolerStat.lrTempColdHead:= Heater_DetIF.Temp.stat.lrTempK - 0.1;
// IF cooler.in_bEnable	THEN
// 	refCoolerStat.bActive	:= TRUE;
// 	refCoolerStat.nDevState	:= E_CRYO_CRYOTELGT_STATE.ON;
// ELSE
// 	refCoolerStat.bActive	:= FALSE;
// 	refCoolerStat.nDevState	:= E_CRYO_CRYOTELGT_STATE.OFF;
// END_IF
END_METHOD

METHOD M_StateMachine
VAR_INPUT
END_VAR
////////////////
// State Machine
////////////////
CASE stat.nState OF
	/////////////////////////////////
	E_NOTT_CRYO_CTRL_STATE.NONE:
	/////////////////////////////////
	//
	// This is the state on power-up.
	// Determine the initial state based on the command and actuator state.
	M_GetState();	
	RETURN;
	

	/////////////////////////////////
	E_NOTT_CRYO_CTRL_STATE.WARM_PRESS:
	/////////////////////////////////
	//
	
	ctrl.bEnable_CoolDown := FALSE;
	ctrl.bEnable_WarmUp   := FALSE;
	
	// Reject any queued top-level sequence command in WARM_PRESS.
	// Evacuation is not handled through ctrl.bExecute / ctrl.nCommand.
	IF ctrl.bExecute THEN
		stat.nLastCommand := ctrl.nCommand;
		ctrl.bExecute     := FALSE;
		ctrl.nCommand     := E_NOTT_CRYO_CTRL_CMD.NONE;
	
		CASE stat.nLastCommand OF
			E_NOTT_CRYO_CTRL_CMD.COOL:
				logs.M_LogInfo('COOL command rejected: system is WARM_PRESS. Evacuate first.');
	
			E_NOTT_CRYO_CTRL_CMD.WARM_UP:
				logs.M_LogInfo('WARM_UP command rejected: system is already warm pressurized.');
		ELSE
				logs.M_LogInfo('Command rejected: system is WARM_PRESS.');
		END_CASE
	END_IF
	
	// Evacuation itself is not part of this state machine.
	// Once pressure status says the cryostat is in vacuum, recover to WARM_VACUUM.
	IF stat.bVacuumOK OR stat.bVacuum THEN
		ctrl.bEnable_CoolDown := FALSE;
		ctrl.bEnable_WarmUp   := FALSE;
	
		logs.M_LogInfo('Vacuum detected. State is WARM_VACUUM.');
		stat.nState := E_NOTT_CRYO_CTRL_STATE.WARM_VACUUM;
	END_IF
	
	M_SetStatus(stat.nState);
	RETURN;
	
	
	//////////////////////////////////////////
	E_NOTT_CRYO_CTRL_STATE.WARM_VACUUM:
	//////////////////////////////////////////
	//
		
		// Keep warmup inactive unless a permitted WARM_UP command is accepted.
		ctrl.bEnable_WarmUp := FALSE;
		
		// If the system is already cold/operational, recover to COLD.
		IF stat.bOP OR stat.bCold THEN
			ctrl.bEnable_Evac := TRUE;
		
			logs.M_LogInfo('Cold condition detected. State is COLD.');
			stat.nState := E_NOTT_CRYO_CTRL_STATE.COLD;
		
		// If vacuum is lost, return to WARM_PRESS.
		ELSIF NOT (stat.bVacuumOK OR stat.bVacuum) THEN
			ctrl.bEnable_CoolDown := FALSE;
			ctrl.bEnable_WarmUp   := FALSE;
		
			logs.M_LogInfo('Vacuum lost. State is WARM_PRESS.');
			stat.nState := E_NOTT_CRYO_CTRL_STATE.WARM_PRESS;
		
		// Process queued top-level commands.
		ELSIF ctrl.bExecute THEN
			ctrl.bExecute     := FALSE;
			stat.nLastCommand := ctrl.nCommand;
			ctrl.nCommand     := E_NOTT_CRYO_CTRL_CMD.NONE;
		
			CASE stat.nLastCommand OF
		
				E_NOTT_CRYO_CTRL_CMD.COOL:
					// Cool down only if top-level permissions and cooler state allow it.
					IF cool_down.bPermitStart AND cool_down.cooler.stat.bInitialised THEN
						logs.M_LogInfo('Cool-down started.');
		
						ctrl.bEnable_Evac     := TRUE;
						ctrl.bEnable_CoolDown := TRUE;
						ctrl.bEnable_WarmUp   := FALSE;
		
						stat.nState := E_NOTT_CRYO_CTRL_STATE.COOLING_DOWN;
					ELSIF NOT cool_down.bPermitStart THEN
						ctrl.bEnable_CoolDown := FALSE;
						logs.M_LogInfo('COOL command rejected: cooldown start not permitted.');
					ELSE
						ctrl.bEnable_CoolDown := FALSE;
						logs.M_LogInfo('COOL command rejected: cooler not initialised.');
					END_IF
		
				E_NOTT_CRYO_CTRL_CMD.WARM_UP:
					// Normally not allowed in WARM_VACUUM by the current permission table.
					IF warm_up.bPermitStart THEN
						logs.M_LogInfo('Warm-up started.');
		
						ctrl.bEnable_Evac     := TRUE;
						ctrl.bEnable_WarmUp   := TRUE;
						ctrl.bEnable_CoolDown := FALSE;
		
						stat.nState := E_NOTT_CRYO_CTRL_STATE.WARMING_UP;
					ELSE
						ctrl.bEnable_WarmUp := FALSE;
						logs.M_LogInfo('WARM_UP command rejected: warmup start not permitted in WARM_VACUUM.');
					END_IF
		
			ELSE
				logs.M_LogInfo('Command rejected: unsupported command in WARM_VACUUM.');
			END_CASE
		END_IF
		
		M_SetStatus(stat.nState);
		RETURN;
	

	///////////////////////////////////
	E_NOTT_CRYO_CTRL_STATE.COOLING_DOWN:
	///////////////////////////////////
	//
	
	// Evacuation should remain enabled during cooldown.
	ctrl.bEnable_Evac := TRUE;
	
	// Reject queued top-level sequence commands while cooldown is active.
	// Stop cooldown via ctrl.bEnable_CoolDown FALSE and permission logic.
	IF ctrl.bExecute THEN
		stat.nLastCommand := ctrl.nCommand;
		ctrl.bExecute     := FALSE;
		ctrl.nCommand     := E_NOTT_CRYO_CTRL_CMD.NONE;
	
		CASE stat.nLastCommand OF
			E_NOTT_CRYO_CTRL_CMD.COOL:
				logs.M_LogInfo('COOL command ignored: cooldown already active.');
	
			E_NOTT_CRYO_CTRL_CMD.WARM_UP:
				logs.M_LogInfo('WARM_UP command rejected: cooldown active.');
		ELSE
				logs.M_LogInfo('Command rejected: cooldown active.');
		END_CASE
	END_IF
	
	// Operational or cold condition reached.
	IF stat.bOP OR stat.bCold THEN
		ctrl.bEnable_Evac := TRUE;
	
		logs.M_LogInfo('Cold/operational condition reached. State is COLD.');
		stat.nState := E_NOTT_CRYO_CTRL_STATE.COLD;
	
	// Vacuum lost during cooldown.
	ELSIF NOT (stat.bVacuumOK OR stat.bVacuum) THEN
		ctrl.bEnable_CoolDown := FALSE;
		ctrl.bEnable_WarmUp   := FALSE;
	
		logs.M_LogInfo('Vacuum lost during cooldown. State is WARM_PRESS.');
		stat.nState := E_NOTT_CRYO_CTRL_STATE.WARM_PRESS;
	
	// Cooldown stopped by command/permission.
	ELSIF NOT ctrl.bEnable_CoolDown THEN
		ctrl.bEnable_WarmUp := FALSE;
	
		IF stat.bVacuumOK OR stat.bVacuum THEN
			logs.M_LogInfo('Cooldown stopped. State is WARM_VACUUM.');
			stat.nState := E_NOTT_CRYO_CTRL_STATE.WARM_VACUUM;
		ELSE
			logs.M_LogInfo('Cooldown stopped and vacuum not present. State is WARM_PRESS.');
			stat.nState := E_NOTT_CRYO_CTRL_STATE.WARM_PRESS;
		END_IF
	
	// Once startup has completed, an inactive cooler is unexpected. Do not
	// apply this check in START_PTC while the cooler is still starting.
	ELSIF ((cool_down.stat.nState = E_NOTT_CRYO_COOLDOWN_STATE.COOLING)
		OR (cool_down.stat.nState = E_NOTT_CRYO_COOLDOWN_STATE.OPERATIONAL_TEMPERATURE_ACHIEVED))
		AND NOT cool_down.cooler.stat.bActive THEN
		ctrl.bEnable_CoolDown := FALSE;
		ctrl.bEnable_WarmUp   := FALSE;
	
		IF stat.bVacuumOK OR stat.bVacuum THEN
			logs.M_LogInfo('Cooler inactive. State is WARM_VACUUM.');
			stat.nState := E_NOTT_CRYO_CTRL_STATE.WARM_VACUUM;
		ELSE
			logs.M_LogInfo('Cooler inactive and vacuum not present. State is WARM_PRESS.');
			stat.nState := E_NOTT_CRYO_CTRL_STATE.WARM_PRESS;
		END_IF
	END_IF
	
	M_SetStatus(stat.nState);
	RETURN;
	
	
	///////////////////////////////////////////
	E_NOTT_CRYO_CTRL_STATE.COLD:
	///////////////////////////////////////////

		// While operational, preserve the operator's evacuation command. If OP is
		// lost after evacuation was stopped, restart evacuation and cooldown once
		// on the filtered OP falling edge.
		IF triggers.OP_OFF.Q AND NOT evac.bEvacuationActive THEN
			ctrl.bEnable_Evac     := TRUE;
			ctrl.bEnable_CoolDown := TRUE;
			ctrl.bEnable_WarmUp   := FALSE;

			logs.M_LogInfo('Operational state lost with evacuation inactive. Restarting evacuation and cooldown.');
			stat.nState := E_NOTT_CRYO_CTRL_STATE.COOLING_DOWN;
		END_IF
		
